REGION Network 2: +++ Werkingsmode Hand +++
   // Verwerking van de bedieningen van het aanraakscherm, en bepalen van de bedieningsmode Hand.
END_REGION

REGION Network 3: +++ Gewenste stand +++
   // Bepalen aan de hand van de actuele bediening of ontvangen sturing, wat de gewenste stand van de klep is.
END_REGION

REGION Network 4: +++ Klepsturing +++
   // Aansturen van de klep en terugmeldingsbewaking.
END_REGION

REGION Network 5: +++ Storingen +++
   // Verwerken van de storingsmeldingen.
END_REGION

REGION Network 6: Storing A001: Beveiliging aangesproken
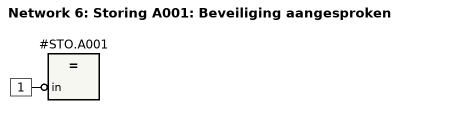
   #STO.A001 := NOT 1;
END_REGION

REGION Network 7 (SCL): EINDE
   // Variabelen van intern scada rakvlak naar outputs copieren
   #VAR_IF_KLG.STS_OPEN := #VAR.STS_OPEN;
   #VAR_IF_KLG.STS_TOE := #VAR.STS_TOE;
   #VAR_IF_KLG.STS_BEZ_OPEN := #VAR.STS_BEZ_OPEN;
   #VAR_IF_KLG.STS_BEZ_TOE := #VAR.STS_BEZ_TOE;
   #VAR_IF_KLG.BMO_HAND := #VAR.BMO_HAND;
   #VAR_IF_KLG.EXT_HW := #VAR.EXT_HW;
   #VAR_IF_KLG.STO := #STO;
END_REGION
END_FUNCTION_BLOCK

FUNCTION_BLOCK "TYPIC_C501_IF_KLH"   // FB63, FBD
TITLE = TYPIC_C501_IF_KLH: Handbediende klep
{ S7_Optimized_Access := 'TRUE' }
AUTHOR : OCOTECH
FAMILY : Typical
NAME : C501.704
// Logisch Object Besturing: C501.704
// 
// De interne functie handbediende klep verzorgt de bewaking van één van volgende componenten:
//  een handbediende klep
//  een leegzetvoorziening
//  een beo/ontluchtingsvoorziening
// stored: MemoryReserve 10, SetENOAutomatically false
   VAR_INPUT
      EXT_HW { ExternalAccessible := 'False'; ExternalVisible := 'False'; ExternalWritable := 'False'} : Bool;   // Sturings hardware (PLC) bewaking (1 = OK)
      IN_OPEN { ExternalAccessible := 'False'; ExternalVisible := 'False'; ExternalWritable := 'False'} : Bool;   // Handbediende klep is open
      IN_TOE { ExternalAccessible := 'False'; ExternalVisible := 'False'; ExternalWritable := 'False'} : Bool;   // Handbediende klep is toe
      CFG_OPEN { ExternalAccessible := 'False'; ExternalVisible := 'False'; ExternalWritable := 'False'} : Bool;   // Handbediende klep heeft een toestandsmelding Open
      CFG_TOE { ExternalAccessible := 'False'; ExternalVisible := 'False'; ExternalWritable := 'False'} : Bool;   // Handbediende klep heeft een toestandsmelding Toe
   END_VAR
   VAR_OUTPUT
      VAR_IF_KLH { ExternalAccessible := 'False'; ExternalVisible := 'False'; ExternalWritable := 'False'} : "C501_VAR_IF_KLH_TYPIC";   // Struct met alle variabelen naar bovenliggende functies
   END_VAR
   VAR
      STO { ExternalWritable := 'False'} : Struct   // Storingen
         A001 : Bool;   // Terugmeldingen Open en Dicht tegelijk
      END_STRUCT;
      VAR { ExternalWritable := 'False'} : Struct   // Variabelen
         STS_OPEN : Bool;   // Handbediende klep is open
         STS_TOE : Bool;   // Handbediende klep is toe
         EXT_HW { ExternalAccessible := 'False'; ExternalVisible := 'False'} : Bool;   // Sturings hardware (PLC) in storing
      END_STRUCT;
   END_VAR
BEGIN

REGION Network 1: START
END_REGION

REGION Network 2: +++ Status +++
   // De status van de handbediende klep (open / dicht) wordt doorgestuurd naar 3B.
END_REGION

REGION Network 3: +++ Storingen +++
   // Alle storingen worden doorgegeven aan 3B.
END_REGION

REGION Network 4: Storing A001: Terugmeldingen Open en Dicht tegelijk
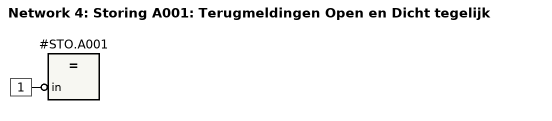
   #STO.A001 := NOT 1;
END_REGION

REGION Network 5 (SCL): EINDE
   // Variabelen van intern scada rakvlak naar outputs copieren
   #VAR_IF_KLH.STS_OPEN := #VAR.STS_OPEN;
   #VAR_IF_KLH.STS_TOE := #VAR.STS_TOE;
   #VAR_IF_KLH.EXT_HW := #VAR.EXT_HW;
   #VAR_IF_KLH.STO := #STO;
END_REGION
END_FUNCTION_BLOCK

FUNCTION_BLOCK "TYPIC_C501_IF_NME"   // FB62, FBD
TITLE = TYPIC_C501_IF_NME: Niveaumeting
{ S7_Optimized_Access := 'TRUE' }
AUTHOR : OCOTECH
FAMILY : Typical
NAME : C501.702
// Logisch Object Besturing: C501.702
// 
// De interne functie niveaumeting verzorgt de interne besturing en bewaking van een niveaumeting van de brandblusinstallatie.
// stored: MemoryReserve 10, SetENOAutomatically false
   VAR_INPUT
      EXT_HW { ExternalAccessible := 'False'; ExternalVisible := 'False'; ExternalWritable := 'False'} : Bool;   // Sturings hardware (PLC) bewaking (1 = OK)
      IN_MWA { ExternalAccessible := 'False'; ExternalVisible := 'False'; ExternalWritable := 'False'} : Word;   // Meetwaarde
      IN_HW { ExternalAccessible := 'False'; ExternalVisible := 'False'; ExternalWritable := 'False'} : Bool;   // Vlotter: 1 = Bovenwater / 0 = Onderwater
      IN_VHW { ExternalAccessible := 'False'; ExternalVisible := 'False'; ExternalWritable := 'False'} : Bool;   // Vlotter: 1 = Bovenwater / 0 = Onderwater
      IN_SD { ExternalAccessible := 'False'; ExternalVisible := 'False'; ExternalWritable := 'False'} : Bool;   // Vlotter: 1 = Bovenwater / 0 = Onderwater
      IN_SO { ExternalAccessible := 'False'; ExternalVisible := 'False'; ExternalWritable := 'False'} : Bool;   // Vlotter: 1 = Onderwater / 0 = Bovenwater
      IN_VRL { ExternalAccessible := 'False'; ExternalVisible := 'False'; ExternalWritable := 'False'} : Bool;   // Vlotter: 1 = Onderwater / 0 = Bovenwater
      IN_RL { ExternalAccessible := 'False'; ExternalVisible := 'False'; ExternalWritable := 'False'} : Bool;   // Vlotter: 1 = Onderwater / 0 = Bovenwater
      IN_AUT_C501 { ExternalAccessible := 'False'; ExternalVisible := 'False'; ExternalWritable := 'False'} : Bool;   // Beveiligingen: serie geschakelde terugmelding (1= OK)
      CFG_MAX { ExternalAccessible := 'False'; ExternalVisible := 'False'; ExternalWritable := 'False'} : Int;   // Waarde van input IN_MWA als maximum voor de scalering ter bepaling van NIV_MWA
      CFG_MIN { ExternalAccessible := 'False'; ExternalVisible := 'False'; ExternalWritable := 'False'} : Int;   // Waarde van input IN_MWA als minimum voor de scalering ter bepaling van NIV_MWA
      CFG_MAX_SWA { ExternalAccessible := 'False'; ExternalVisible := 'False'; ExternalWritable := 'False'} : Real;   // Waarde die toegekend wordt aan NIV_MWA als maximumwmaximumwaarde voor de meeteenheid
      CFG_MIN_SWA { ExternalAccessible := 'False'; ExternalVisible := 'False'; ExternalWritable := 'False'} : Real;   // Waarde die toegekend wordt aan NIV_MWA als minimumwmaximumwaarde voor de meeteenheid
   END_VAR
   VAR_OUTPUT
      VAR_IF_NME { ExternalAccessible := 'False'; ExternalVisible := 'False'; ExternalWritable := 'False'} : "C501_VAR_IF_NME_TYPIC";   // Struct met alle variabelen naar de basisfunctie
   END_VAR
   VAR
      STO { ExternalWritable := 'False'} : Struct   // Storingen
         A001 : Bool;   // Beveiliging aangesproken
         A002 : Bool;   // Draadbreuk analoge meting
         A003 : Bool;   // Meetbereik overschreden
         A004 : Bool;   // Status vlotters inconsistent
      END_STRUCT;
      VAR { ExternalWritable := 'False'} : Struct   // Variabelen
         MWA : Real;   // Meetwaarde
         HW : USInt;   // Hoogwater vlotter
         VHW : USInt;   // Voorwaarschuwing hoogwater
         SD : USInt;   // Suppletie dicht
         SO : USInt;   // Suppletie open
         VRL : USInt;   // Voorwaarschuwing reservoir leeg
         RL : USInt;   // Reservoir leeg
         EXT_HW { ExternalAccessible := 'False'; ExternalVisible := 'False'} : Bool;   // Sturings hardware (PLC) in storing
      END_STRUCT;
   END_VAR
BEGIN

REGION Network 1: START
END_REGION

REGION Network 2: +++ Bepalen status peilen (vlotters) +++
   // Aan de hand van de status van de vlotters (inputs) wordt het peil (onderwater/bovenwater) bepaalt.
END_REGION

REGION Network 3: +++ Meting +++
   // Verwerken van de analoge meting.
END_REGION

REGION Network 4: +++ Storingen +++
   // Verwerken van de storingsmeldingen.
END_REGION

REGION Network 5: Storing A001: Beveiliging aangesproken
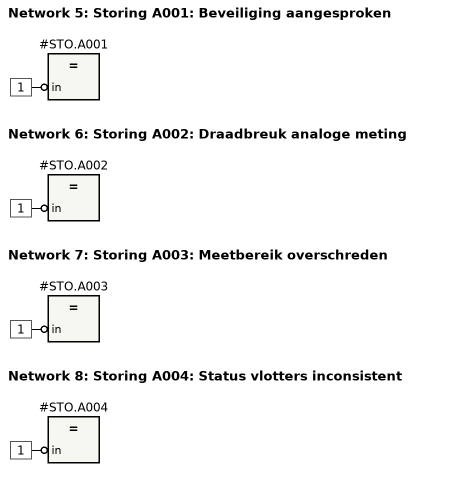
   #STO.A001 := NOT 1;
END_REGION

REGION Network 6: Storing A002: Draadbreuk analoge meting
   #STO.A002 := NOT 1;
END_REGION

REGION Network 7: Storing A003: Meetbereik overschreden
   #STO.A003 := NOT 1;
END_REGION

REGION Network 8: Storing A004: Status vlotters inconsistent
   #STO.A004 := NOT 1;
END_REGION

REGION Network 9 (SCL): EINDE
   // Variabelen van intern scada rakvlak naar outputs copieren
   #VAR_IF_NME.MWA := #VAR.MWA;
   #VAR_IF_NME.HW := #VAR.HW;
   #VAR_IF_NME.VHW := #VAR.VHW;
   #VAR_IF_NME.SD := #VAR.SD;
   #VAR_IF_NME.SO := #VAR.SO;
   #VAR_IF_NME.VRL := #VAR.VRL;
   #VAR_IF_NME.RL := #VAR.RL;
   #VAR_IF_NME.EXT_HW := #VAR.EXT_HW;
   #VAR_IF_NME.STO := #STO;
END_REGION
END_FUNCTION_BLOCK

FUNCTION_BLOCK "TYPIC_C501_IF_SME"   // FB61, FBD
TITLE = TYPIC_C501_IF_SME: Debietmeting
{ S7_Optimized_Access := 'TRUE' }
AUTHOR : OCOTECH
FAMILY : Typical
NAME : C501.711
// Logisch Object Besturing: C501.711
// 
// De interne functie debietmeting verzorgt de interne besturing en bewaking van een debietmeting.
// stored: MemoryReserve 10, SetENOAutomatically false
   VAR_INPUT
      EXT_HW { ExternalAccessible := 'False'; ExternalVisible := 'False'; ExternalWritable := 'False'} : Bool;   // Sturings hardware (PLC) bewaking (1 = OK)
      IN_MWA { ExternalAccessible := 'False'; ExternalVisible := 'False'; ExternalWritable := 'False'} : Word;   // Meetwaarde
      IN_STO { ExternalAccessible := 'False'; ExternalVisible := 'False'; ExternalWritable := 'False'} : Bool;   // Storing (1= OK)
      IN_AUT_C501 { ExternalAccessible := 'False'; ExternalVisible := 'False'; ExternalWritable := 'False'} : Bool;   // Beveiligingen: serie geschakelde terugmelding (1= OK)
      CFG_MAX_SWA { ExternalAccessible := 'False'; ExternalVisible := 'False'; ExternalWritable := 'False'} : Real;   // Maximale waarde debietmeting
   END_VAR
   VAR_OUTPUT
      VAR_IF_SME { ExternalAccessible := 'False'; ExternalVisible := 'False'; ExternalWritable := 'False'} : "C501_VAR_IF_SME_TYPIC";   // Struct met alle variabelen naar bovenliggende functies
   END_VAR
   VAR
      STO { ExternalWritable := 'False'} : Struct   // Storingen
         A001 : Bool;   // Beveiliging aangesproken
         A002 : Bool;   // Draadbreuk analoge meting
         A003 : Bool;   // Meetbereik overschreden
         A004 : Bool;   // Debietmeter geeft storing
      END_STRUCT;
      VAR { ExternalWritable := 'False'} : Struct   // Variabelen
         MWA : Real;   // Meetwaarde
         EXT_HW { ExternalAccessible := 'False'; ExternalVisible := 'False'} : Bool;   // Sturings hardware (PLC) in storing
      END_STRUCT;
   END_VAR
BEGIN

REGION Network 1: START
END_REGION

REGION Network 2: +++ Verwerking analoge meting +++
   // Verwerking analoge meting naar een meetwaarde in m3/u en detectie storingen van de meting.
END_REGION

REGION Network 3: +++ Storingen +++
   // Storingen van de analoge meting.
END_REGION

REGION Network 4: Storing A001: Beveiliging aangesproken
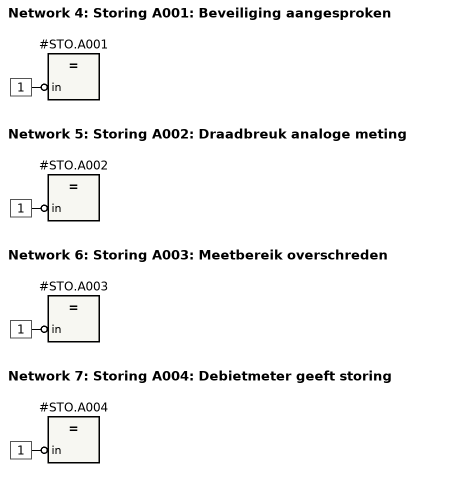
   #STO.A001 := NOT 1;
END_REGION

REGION Network 5: Storing A002: Draadbreuk analoge meting
   #STO.A002 := NOT 1;
END_REGION

REGION Network 6: Storing A003: Meetbereik overschreden
   #STO.A003 := NOT 1;
END_REGION

REGION Network 7: Storing A004: Debietmeter geeft storing
   #STO.A004 := NOT 1;
END_REGION

REGION Network 8 (SCL): EINDE
   // Variabelen van intern scada rakvlak naar outputs copieren
   #VAR_IF_SME.MWA := #VAR.MWA;
   #VAR_IF_SME.EXT_HW := #VAR.EXT_HW;
   #VAR_IF_SME.STO := #STO;
END_REGION
END_FUNCTION_BLOCK

FUNCTION_BLOCK "TYPIC_C501_IF_TME"   // FB60, FBD
TITLE = TYPIC_C501_IF_TME: Temperatuurmeting
{ S7_Optimized_Access := 'TRUE' }
AUTHOR : OCOTECH
FAMILY : Typical
NAME : C501.712
// Logisch Object Besturing: C501.712
// 
// De interne functie temperatuurmeting verzorgt de interne besturing en bewaking van een temperatuurmeting.
// stored: MemoryReserve 10, SetENOAutomatically false
   VAR_INPUT
      EXT_HW { ExternalAccessible := 'False'; ExternalVisible := 'False'; ExternalWritable := 'False'} : Bool;   // Sturings hardware (PLC) bewaking (1 = OK)
      IN_MWA { ExternalAccessible := 'False'; ExternalVisible := 'False'; ExternalWritable := 'False'} : Word;   // Meetwaarde
      IN_AUT_C501 { ExternalAccessible := 'False'; ExternalVisible := 'False'; ExternalWritable := 'False'} : Bool;   // Beveiligingen: serie geschakelde terugmelding (1= OK)
      CFG_MAX_SWA { ExternalAccessible := 'False'; ExternalVisible := 'False'; ExternalWritable := 'False'} : Real;   // Maximale waarde temperatuurmeting
      CFG_MIN_SWA { ExternalAccessible := 'False'; ExternalVisible := 'False'; ExternalWritable := 'False'} : Real;   // Minimale waarde temperatuurmeting
   END_VAR
   VAR_OUTPUT
      VAR_IF_TME { ExternalAccessible := 'False'; ExternalVisible := 'False'; ExternalWritable := 'False'} : "C501_VAR_IF_TME_TYPIC";   // Struct met alle variabelen naar bovenliggende functies
   END_VAR
   VAR
      STO { ExternalWritable := 'False'} : Struct   // Storingen
         A001 : Bool;   // Beveiliging aangesproken
         A002 : Bool;   // Draadbreuk analoge meting
         A003 : Bool;   // Meetbereik overschreden
         A004 : Bool;   // Temperatuurmeter geeft storing
      END_STRUCT;
      VAR { ExternalWritable := 'False'} : Struct   // Variabelen
         MWA : Real;   // Meetwaarde
         EXT_HW { ExternalAccessible := 'False'; ExternalVisible := 'False'} : Bool;   // Sturings hardware (PLC) in storing
      END_STRUCT;
   END_VAR
BEGIN

REGION Network 1: START
END_REGION

REGION Network 2: +++ Verwerking analoge meting +++
   // Verwerking analoge meting naar een meetwaarde in m3/u en detectie storingen van de meting.
END_REGION

REGION Network 3: +++ Storingen +++
   // Storingen van de analoge meting.
END_REGION

REGION Network 4: Storing A001: Beveiliging aangesproken
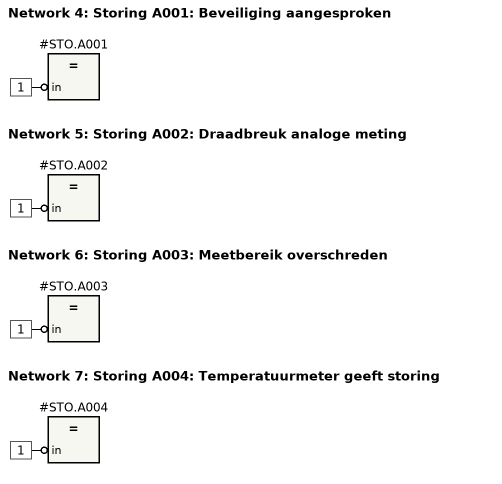
   #STO.A001 := NOT 1;
END_REGION

REGION Network 5: Storing A002: Draadbreuk analoge meting
   #STO.A002 := NOT 1;
END_REGION

REGION Network 6: Storing A003: Meetbereik overschreden
   #STO.A003 := NOT 1;
END_REGION

REGION Network 7: Storing A004: Temperatuurmeter geeft storing
   #STO.A004 := NOT 1;
END_REGION

REGION Network 8 (SCL): EINDE
   // Variabelen van intern scada rakvlak naar outputs copieren
   #VAR_IF_TME.MWA := #VAR.MWA;
   #VAR_IF_TME.EXT_HW := #VAR.EXT_HW;
   #VAR_IF_TME.STO := #STO;
END_REGION
END_FUNCTION_BLOCK

FUNCTION_BLOCK "TYPIC_C501_IF_TRA"   // FB59, FBD
TITLE = TYPIC_C501_IF_TRA: Tracing
{ S7_Optimized_Access := 'TRUE' }
AUTHOR : OCOTECH
FAMILY : Typical
NAME : C501.705
// Logisch Object Besturing: C501.705
// stored: MemoryReserve 10, SetENOAutomatically false
   VAR_INPUT
      EXT_HW { ExternalAccessible := 'False'; ExternalVisible := 'False'; ExternalWritable := 'False'} : Bool;   // Sturings hardware (PLC) bewaking (1 = OK)
      IN_STO { ExternalAccessible := 'False'; ExternalVisible := 'False'; ExternalWritable := 'False'} : Bool;   // Storing Tracing (1 = OK)
   END_VAR
   VAR_OUTPUT
      VAR_IF_TRA { ExternalAccessible := 'False'; ExternalVisible := 'False'; ExternalWritable := 'False'} : "C501_VAR_IF_TRA_TYPIC";   // Struct met alle variabelen naar bovenliggende functies
   END_VAR
   VAR
      STO { ExternalWritable := 'False'} : Struct   // Storingen
         A001 : Bool;   // Storing vorstbeveiliging
      END_STRUCT;
      VAR { ExternalWritable := 'False'} : Struct   // Variabelen
         EXT_HW { ExternalAccessible := 'False'; ExternalVisible := 'False'} : Bool;   // Sturings hardware (PLC) in storing
      END_STRUCT;
   END_VAR
BEGIN

REGION Network 1: START
END_REGION

REGION Network 2: +++ Storingen +++
   // Verwerken van de storingsmeldingen (inputs).
END_REGION

REGION Network 3: Storing A001: Storing vorstbeveiliging
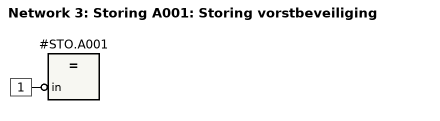
   #STO.A001 := NOT 1;
END_REGION

REGION Network 4 (SCL): EINDE
   // Variabelen van intern scada rakvlak naar outputs copieren
   #VAR_IF_TRA.EXT_HW := #VAR.EXT_HW;
   #VAR_IF_TRA.STO := #STO;
END_REGION
END_FUNCTION_BLOCK

FUNCTION_BLOCK "TYPIC_C501_SF_DME"   // FB55, FBD
TITLE = TYPIC_C501_SF_DME: Drukmeting
{ S7_Optimized_Access := 'TRUE' }
AUTHOR : OCOTECH
FAMILY : Typical
NAME : C501.813
// Logisch Object Besturing: C501.813
// 
// Het doel van deze subfunctie is om de algemene sturing en bediening vanuit 3B te voorzien van een drukmeting behorende tot de brandblusinstallatie.
// stored: MemoryReserve 10, SetENOAutomatically false
   VAR_INPUT
      CFG_SIG_HH { ExternalAccessible := 'False'; ExternalVisible := 'False'; ExternalWritable := 'False'} : Real;   // Schakeldrempel signalering te hoog
      CFG_SIG_H { ExternalAccessible := 'False'; ExternalVisible := 'False'; ExternalWritable := 'False'} : Real;   // Schakeldrempel signalering voorwaarschuwing hoog
      CFG_HYS_H { ExternalAccessible := 'False'; ExternalVisible := 'False'; ExternalWritable := 'False'} : Real;   // Hysteresis op signalering te hoog en voorwaarschuwing hoog
      CFG_ITYD_H { ExternalAccessible := 'False'; ExternalVisible := 'False'; ExternalWritable := 'False'} : Real;   // Tijdsvertraging signalering te hoog
      CFG_SIG_L { ExternalAccessible := 'False'; ExternalVisible := 'False'; ExternalWritable := 'False'} : Real;   // Schakeldrempel signalering te laag
      CFG_HYS_L { ExternalAccessible := 'False'; ExternalVisible := 'False'; ExternalWritable := 'False'} : Real;   // Hysteresis op signalering te laag
      CFG_ITYD_L { ExternalAccessible := 'False'; ExternalVisible := 'False'; ExternalWritable := 'False'} : Time;   // Tijdsvertraging signalering te laag
   END_VAR
   VAR_OUTPUT
      VAR_DME { ExternalAccessible := 'False'; ExternalVisible := 'False'; ExternalWritable := 'False'} : "C501_VAR_DME_TYPIC";   // Struct met alle variabelen van de drukmeting
   END_VAR
   VAR_IN_OUT
      STU_DME : "C501_STU_DME_TYPIC";   // Struct met alle sturingen vanuit de bovenliggende functie
      VAR_IF_DME : "C501_VAR_IF_DME_TYPIC";   // Struct met alle variabelen vanuit de interne sturing
   END_VAR
   VAR
      BED : Struct   // Bedieningen
         OBS : Struct   // Activeer of deactiveer de detectie van de stand van de deur van de hydrantkast
            X : "UDT_BED_ALG";
            KNOP { S7_SetPoint := 'True'} : Array[0..1] of "UDT_BED_KNOP";
         END_STRUCT;
      END_STRUCT;
      BED_OBS { ExternalWritable := 'False'} : "TYPIC_HF_BED_ALG_KNOP";   // Activeer of deactiveer de detectie van de stand van de deur van de hydrantkast
      SIG { ExternalWritable := 'False'} : Struct   // Signaleringen
         AA01 : Bool;   // Drukmeting niet observeerbaar
         AA02 : Bool;   // Storing algemeen
         AA03 : Bool;   // Druk te laag
         AA04 : Bool;   // Voorwaarschuwing druk hoog
         AA05 : Bool;   // Druk te hoog
         A001 : Bool;   // Beveiliging aangesproken
         A002 : Bool;   // Draadbreuk analoge meting
         A003 : Bool;   // Meetbereik overschreden
      END_STRUCT;
      VAR { ExternalWritable := 'False'} : Struct   // Variabelen
         RNO : USInt;   // Reden niet observeerbaar
         AUT : USInt;   // Beveiliging aangesproken
         MWA : USInt;   // Meetwaarde
         OBS { ExternalAccessible := 'False'; ExternalVisible := 'False'} : USInt;   // Observeerbaarheid
      END_STRUCT;
      HF_BST_OBS { ExternalAccessible := 'False'; ExternalVisible := 'False'; ExternalWritable := 'False'} : "TYPIC_HF_BST_OBS";   // Hulp functie besturing
   END_VAR
   // // BED.OBS.KNOP[0] : InDienst
   // // BED.OBS.KNOP[1] : UitDienst
BEGIN

REGION Network 1: START
END_REGION

REGION Network 2: +++ Bedieningen +++
   // Vrijgave en verwerking van de bedieningen (centrale en lokale bediening). De bedienwaardes worden daarna in de verdere deelfunctionaliteiten gebruikt.
END_REGION

REGION Network 3: Knoppen BED_OBS(Activeer of deactiveer de detectie van de stand van de deur van de hydrantkast)
   // Waardes en vrijge van de knoppen BED_OBS
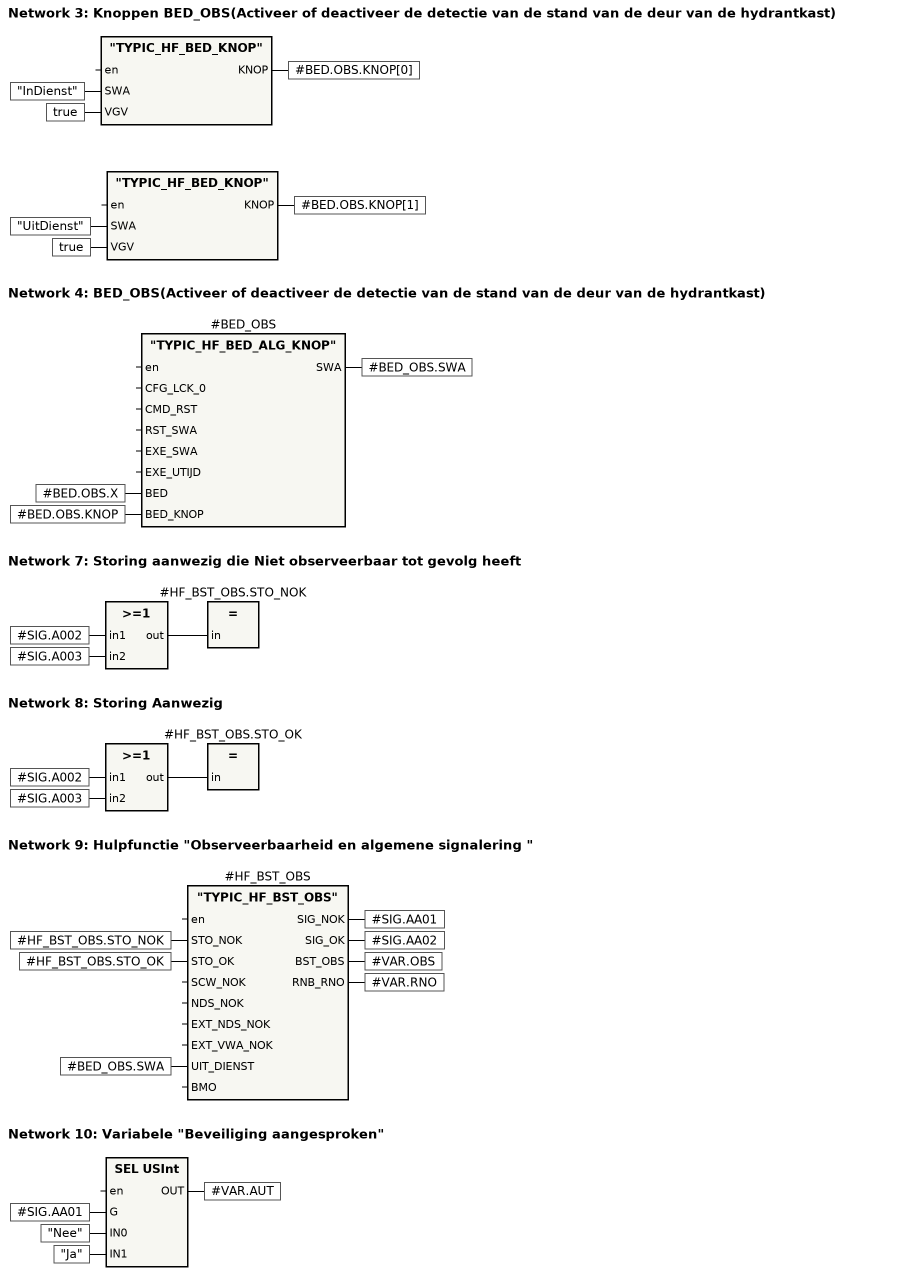
   "TYPIC_HF_BED_KNOP"(SWA := "InDienst", VGV := true, KNOP => #BED.OBS.KNOP[0]);
   "TYPIC_HF_BED_KNOP"(SWA := "UitDienst", VGV := true, KNOP => #BED.OBS.KNOP[1]);
END_REGION

REGION Network 4: BED_OBS(Activeer of deactiveer de detectie van de stand van de deur van de hydrantkast)
   // Verwerking BED_OBS
   #BED_OBS(BED := #BED.OBS.X, BED_KNOP := #BED.OBS.KNOP, SWA => #BED_OBS.SWA);   // "TYPIC_HF_BED_ALG_KNOP"
END_REGION

REGION Network 5: +++ Verwerking meetwaarde en statussen +++
   // De meetwaarde en de status wordt ontvangen vanuit de interne sturing van de drukmeting.
END_REGION

REGION Network 6: +++ Signaleringen en observeerbaarheid +++
   // Aanmaken signaleringen, bepalen observeerbaarheid (observeerbaar / niet observeerbaar) en bepalen reden niet observeerbaar.
END_REGION

REGION Network 7: Storing aanwezig die Niet observeerbaar tot gevolg heeft
   // OR-verknoping van alle storingen om input STO_BST_NOK van de hulpfunctie "Observeerbaarheid en algemene signlaring"
   #HF_BST_OBS.STO_NOK := #SIG.A002 OR #SIG.A003;
END_REGION

REGION Network 8: Storing Aanwezig
   // OR-verknoping van alle storingen om input STO_BST_OK van de hulpfunctie "Observeerbaarheid en algemene signlaring"
   #HF_BST_OBS.STO_OK := #SIG.A002 OR #SIG.A003;
END_REGION

REGION Network 9: Hulpfunctie "Observeerbaarheid en algemene signalering "
   // Bepalen variabele "Observeerbaarheid" en "reden niet Observeerbaarheid", Signaleringen "Observeerbaarheid" en "algmene storing".
   #HF_BST_OBS(STO_NOK := #HF_BST_OBS.STO_NOK,   // "TYPIC_HF_BST_OBS"
               STO_OK := #HF_BST_OBS.STO_OK,
               UIT_DIENST := #BED_OBS.SWA,
               SIG_NOK => #SIG.AA01,
               SIG_OK => #SIG.AA02,
               BST_OBS => #VAR.OBS,
               RNB_RNO => #VAR.RNO);
END_REGION

REGION Network 10: Variabele "Beveiliging aangesproken"
   // De variabele VAR_AUT geef aan of er een beveilliging aangesproken is. Deze variabele laat toe dat de verkeersoperator op SCADA kan zien of er een beveilliging aangesproken is voor deze component.
   #VAR.AUT := SEL(G := #SIG.AA01, IN0 := "Nee", IN1 := "Ja");
END_REGION

REGION Network 11 (SCL): EINDE
   // Variabelen van intern scada rakvlak naar outputs copieren
   #VAR_DME.MWA := #VAR.MWA;
   #VAR_DME.OBS := #VAR.OBS;
END_REGION
END_FUNCTION_BLOCK

FUNCTION_BLOCK "TYPIC_C501_SF_TME"   // FB46, FBD
TITLE = TYPIC_C501_SF_TME: Temperatuurmeting
{ S7_Optimized_Access := 'TRUE' }
AUTHOR : OCOTECH
FAMILY : Typical
NAME : C501.815
// Logisch Object Besturing: C501.815
// 
// Het doel van deze subfunctie is om de algemene sturing en bediening vanuit 3B te voorzien van een temperatuurmeting behorende tot de brandblusinstallatie.
// stored: MemoryReserve 10, SetENOAutomatically false
   VAR_INPUT
      CFG_SIG_L { ExternalAccessible := 'False'; ExternalVisible := 'False'; ExternalWritable := 'False'} : Real;   // Schakeldrempel signalering te laag
      CFG_HYS_L { ExternalAccessible := 'False'; ExternalVisible := 'False'; ExternalWritable := 'False'} : Real;   // Hysteresis op signalering te laag
      CFG_ITYD_L { ExternalAccessible := 'False'; ExternalVisible := 'False'; ExternalWritable := 'False'} : Time;   // Tijdsvertraging signalering te laag
   END_VAR
   VAR_OUTPUT
      VAR_TME { ExternalAccessible := 'False'; ExternalVisible := 'False'; ExternalWritable := 'False'} : "C501_VAR_TME_TYPIC";   // Struct met alle variabelen van de temperatuurmeting
   END_VAR
   VAR_IN_OUT
      STU_TME : "C501_STU_TME_TYPIC";   // Struct met alle sturingen vanuit de bovenliggende functie
      VAR_IF_TME : "C501_VAR_IF_TME_TYPIC";   // Struct met alle variabelen vanuit de interne sturing
   END_VAR
   VAR
      BED : Struct   // Bedieningen
         OBS : Struct   // Activeer of deactiveer de detectie van de stand van de deur van de hydrantkast
            X : "UDT_BED_ALG";
            KNOP { S7_SetPoint := 'True'} : Array[0..1] of "UDT_BED_KNOP";
         END_STRUCT;
      END_STRUCT;
      BED_OBS { ExternalWritable := 'False'} : "TYPIC_HF_BED_ALG_KNOP";   // Activeer of deactiveer de detectie van de stand van de deur van de hydrantkast
      SIG { ExternalWritable := 'False'} : Struct   // Signaleringen
         AA01 : Bool;   // Temperatuurmeting niet observeerbaar
         AA02 : Bool;   // Storing algemeen
         AA03 : Bool;   // Temperatuur te laag
         A001 : Bool;   // Beveiliging aangesproken
         A002 : Bool;   // Draadbreuk analoge meting
         A003 : Bool;   // Meetbereik overschreden
      END_STRUCT;
      VAR { ExternalWritable := 'False'} : Struct   // Variabelen
         RNO : USInt;   // Reden niet observeerbaar
         AUT : USInt;   // Beveiliging aangesproken
         MWA : USInt;   // Meetwaarde
         OBS { ExternalAccessible := 'False'; ExternalVisible := 'False'} : USInt;   // Observeerbaarheid
      END_STRUCT;
      HF_BST_OBS { ExternalAccessible := 'False'; ExternalVisible := 'False'; ExternalWritable := 'False'} : "TYPIC_HF_BST_OBS";   // Hulp functie besturing
   END_VAR
   // // BED.OBS.KNOP[0] : InDienst
   // // BED.OBS.KNOP[1] : UitDienst
BEGIN

REGION Network 1: START
END_REGION

REGION Network 2: +++ Bedieningen +++
   // Vrijgave en verwerking van de bedieningen (centrale en lokale bediening). De bedienwaardes worden daarna in de verdere deelfunctionaliteiten gebruikt.
END_REGION

REGION Network 3: Knoppen BED_OBS(Activeer of deactiveer de detectie van de stand van de deur van de hydrantkast)
   // Waardes en vrijge van de knoppen BED_OBS
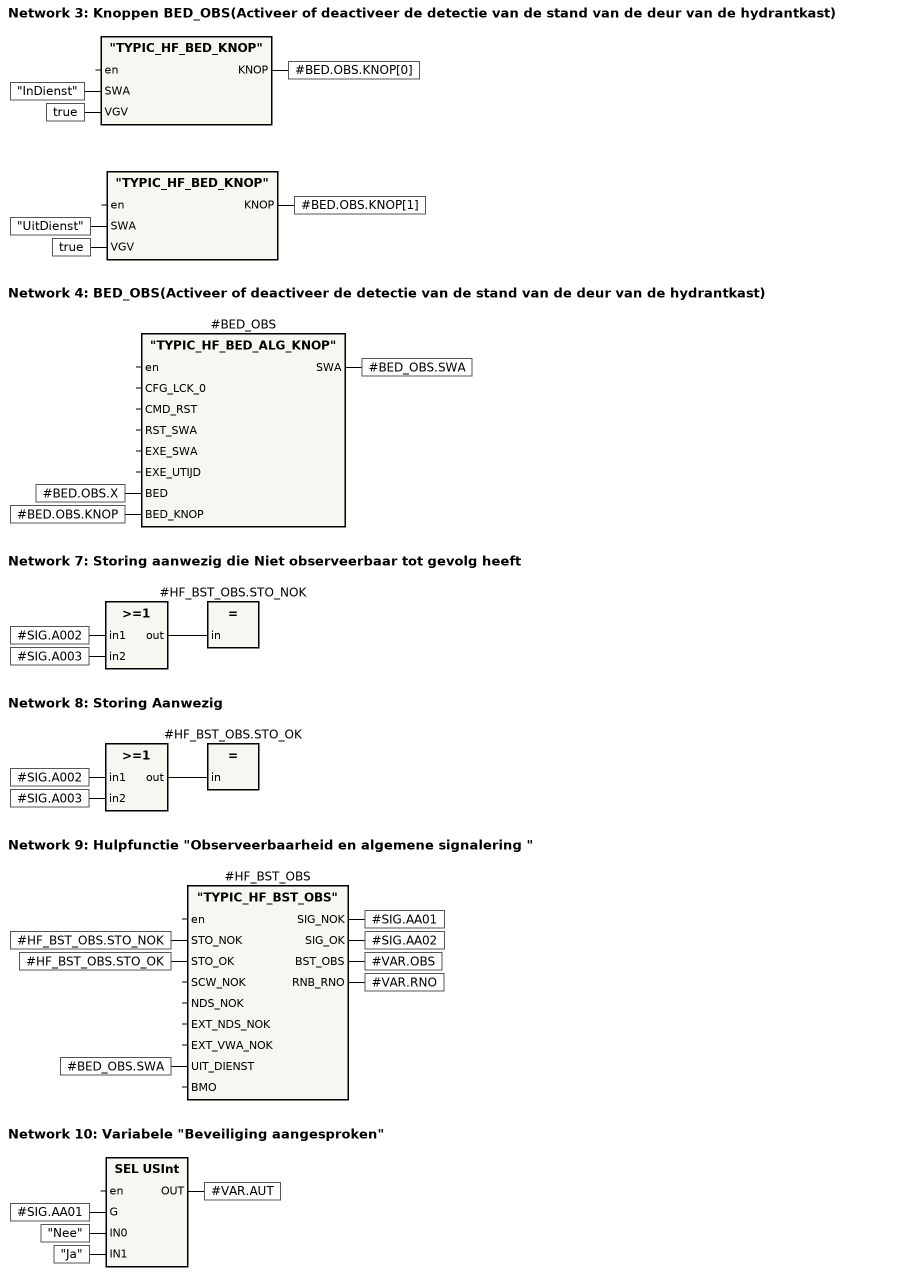
   "TYPIC_HF_BED_KNOP"(SWA := "InDienst", VGV := true, KNOP => #BED.OBS.KNOP[0]);
   "TYPIC_HF_BED_KNOP"(SWA := "UitDienst", VGV := true, KNOP => #BED.OBS.KNOP[1]);
END_REGION

REGION Network 4: BED_OBS(Activeer of deactiveer de detectie van de stand van de deur van de hydrantkast)
   // Verwerking BED_OBS
   #BED_OBS(BED := #BED.OBS.X, BED_KNOP := #BED.OBS.KNOP, SWA => #BED_OBS.SWA);   // "TYPIC_HF_BED_ALG_KNOP"
END_REGION

REGION Network 5: +++ Verwerking meetwaarde en statussen +++
   // De meetwaarde en de status wordt ontvangen vanuit de interne sturing van de temperatuurmeting.
END_REGION

REGION Network 6: +++ Signaleringen en observeerbaarheid +++
   // Aanmaken signaleringen, bepalen observeerbaarheid (observeerbaar / niet observeerbaar) en bepalen reden niet observeerbaar.
END_REGION

REGION Network 7: Storing aanwezig die Niet observeerbaar tot gevolg heeft
   // OR-verknoping van alle storingen om input STO_BST_NOK van de hulpfunctie "Observeerbaarheid en algemene signlaring"
   #HF_BST_OBS.STO_NOK := #SIG.A002 OR #SIG.A003;
END_REGION

REGION Network 8: Storing Aanwezig
   // OR-verknoping van alle storingen om input STO_BST_OK van de hulpfunctie "Observeerbaarheid en algemene signlaring"
   #HF_BST_OBS.STO_OK := #SIG.A002 OR #SIG.A003;
END_REGION

REGION Network 9: Hulpfunctie "Observeerbaarheid en algemene signalering "
   // Bepalen variabele "Observeerbaarheid" en "reden niet Observeerbaarheid", Signaleringen "Observeerbaarheid" en "algmene storing".
   #HF_BST_OBS(STO_NOK := #HF_BST_OBS.STO_NOK,   // "TYPIC_HF_BST_OBS"
               STO_OK := #HF_BST_OBS.STO_OK,
               UIT_DIENST := #BED_OBS.SWA,
               SIG_NOK => #SIG.AA01,
               SIG_OK => #SIG.AA02,
               BST_OBS => #VAR.OBS,
               RNB_RNO => #VAR.RNO);
END_REGION

REGION Network 10: Variabele "Beveiliging aangesproken"
   // De variabele VAR_AUT geef aan of er een beveilliging aangesproken is. Deze variabele laat toe dat de verkeersoperator op SCADA kan zien of er een beveilliging aangesproken is voor deze component.
   #VAR.AUT := SEL(G := #SIG.AA01, IN0 := "Nee", IN1 := "Ja");
END_REGION

REGION Network 11 (SCL): EINDE
   // Variabelen van intern scada rakvlak naar outputs copieren
   #VAR_TME.MWA := #VAR.MWA;
   #VAR_TME.OBS := #VAR.OBS;
END_REGION
END_FUNCTION_BLOCK

FUNCTION_BLOCK "TYPIC_C904_BF_SPI"   // FB44, FBD
TITLE = TYPIC_C904_BF_SPI: Schoonvloeistofpompinstallatie
{ S7_Optimized_Access := 'TRUE' }
AUTHOR : OCOTECH
FAMILY : Typical
NAME : C904.801
// Logisch Object Besturing: C904.801
// 
// 								Het doel van de BF SPI (schoonvloeistofpompinstallatie) is om de
// 								algemene sturing te voorzien van de schoonvloeistofpompinstallatie.
// 								De algemene sturing omvat het weergeven van de algemene toestand en
// 								het aano en afschakelen van pompen in functie van het vloeistofpeil
// 								en het actieve regime.
// stored: MemoryReserve 10, SetENOAutomatically false
   VAR_INPUT
      CFG_TST_UTYD { ExternalAccessible := 'False'; ExternalVisible := 'False'; ExternalWritable := 'False'} : Time;   // Time-out standverandering pompinstallatie (transitiestatus onbereikt)
      CFG_TST_OK_TYD { ExternalAccessible := 'False'; ExternalVisible := 'False'; ExternalWritable := 'False'} : Time;   // Stabilisatietijd voor de toestand OK (bereikt)
      CFG_NIV_H { ExternalAccessible := 'False'; ExternalVisible := 'False'; ExternalWritable := 'False'} : Real;   // Grenswaarde voor dreigende overloop (minder dan 30m3 bergruimte)
      CFG_NIV_HH { ExternalAccessible := 'False'; ExternalVisible := 'False'; ExternalWritable := 'False'} : Real;   // Grenswaarde voor overloop
      CFG_NIV_ITYD { ExternalAccessible := 'False'; ExternalVisible := 'False'; ExternalWritable := 'False'} : Time;   // Inschakelvertraging storingen grenswaarde
      CFG_NIV_HYS { ExternalAccessible := 'False'; ExternalVisible := 'False'; ExternalWritable := 'False'} : Real;   // Hysteresis storingen grenswaarde
      CFG_DEB_H { ExternalAccessible := 'False'; ExternalVisible := 'False'; ExternalWritable := 'False'} : Real;   // Grenswaarde minimaal debiet bij 1 aangeschakelde pomp
      CFG_DEB_HH { ExternalAccessible := 'False'; ExternalVisible := 'False'; ExternalWritable := 'False'} : Real;   // Grenswaarde minimaal debiet bij meerdere aangeschakelde pompen
      CFG_ITYD_DEB { ExternalAccessible := 'False'; ExternalVisible := 'False'; ExternalWritable := 'False'} : Time;   // Tijdsvertraging voor alarm afvoer verstopt (pomp aangeschakeld en minimaal debiet niet bereikt)
      STU_CMD_AUT { ExternalAccessible := 'False'; ExternalVisible := 'False'; ExternalWritable := 'False'} : USInt;   // Groepscommando: schakel in automatisch
      STU_CMD_WRE { ExternalAccessible := 'False'; ExternalVisible := 'False'; ExternalWritable := 'False'} : USInt;   // Sturing regime
      STU_ALG_LCK_SIG { ExternalAccessible := 'False'; ExternalVisible := 'False'; ExternalWritable := 'False'} : USInt;   // Onderdruk alarmen
   END_VAR
   VAR_OUTPUT
      VAR_PWR { ExternalAccessible := 'False'; ExternalVisible := 'False'; ExternalWritable := 'False'} : Real;   // Som actuele vermogens van alle pompen
      STU_PMP1 { ExternalAccessible := 'False'; ExternalVisible := 'False'; ExternalWritable := 'False'} : USInt;   // Sturing pomp
      STU_PMP2 { ExternalAccessible := 'False'; ExternalVisible := 'False'; ExternalWritable := 'False'} : USInt;   // Sturing pomp
      STU_PMP3 { ExternalAccessible := 'False'; ExternalVisible := 'False'; ExternalWritable := 'False'} : USInt;   // Sturing pomp
      STU_IF_SPI { ExternalAccessible := 'False'; ExternalVisible := 'False'; ExternalWritable := 'False'} : USInt;   // Gewenst regime (naar interne sturing)
   END_VAR
   VAR_IN_OUT
      VAR_IF_SPI : "C904_VAR_IF_SPI_TYPIC";   // Struct met variabelen ontvangen van de interne sturing van de pompinstallatie
      VAR_PMP : Array[*] of "C904_VAR_PMP_TYPIC";   // Array met alle pompen, met alle variabelen van de pomp
      VAR_NIV : "C904_VAR_NIV_TYPIC";   // Struct met alle variabelen ontvangen van de subfunctie niveaumeting
      VAR_DEB : "C904_VAR_DEB_TYPIC";   // Struct met alle variabelen ontvangen van de subfunctie debietmeting
   END_VAR
   VAR
      BED : Struct   // Bedieningen
         ALG : Struct   // Gewenste stand
            X : "UDT_BED_ALG";
            KNOP { S7_SetPoint := 'True'} : Array[0..3] of "UDT_BED_KNOP";
         END_STRUCT;
      END_STRUCT;
      BED_ALG { ExternalWritable := 'False'} : "TYPIC_HF_BED_ALG_KNOP";   // Gewenste stand
      SIG { ExternalWritable := 'False'} : Struct   // Signaleringen
         AA01 : Bool;   // Gewenste stand niet bereikt (transitiestatus = niet bereikt)
         AA02 : Bool;   // Schoonvloeistofpompinstallatie dreigt over te lopen
         AA03 : Bool;   // Overschrijding capaciteit schoonvloeistofpompinstallatie (overloop)
         AA04 : Bool;   // Afvoer verstopt en dreiging overloop van de schoonvloeistofpompinstallatie
         AA05 : Bool;   // Afvoer verstopt
         AB01 : Bool;   // Schoonvloeistofpompinstallatie niet beschikbaar
         AB02 : Bool;   // Schoonvloeistofpompinstallatie beperkt beschikbaar
         A001 : Bool;   // Beveiliging aangesproken
         A002 : Bool;   // Beveiliging No-Break aangesproken
         A003 : Bool;   // Overspanningsbeveiliging aangesproken
         A004 : Bool;   // Schuif ALSB uitgeschakeld
         A005 : Bool;   // Schuif ALSB in test
         A006 : Bool;   // Schuif ALSB uitgereden
         A007 : Bool;   // Nisdeur niet gesloten
         A008 : Bool;   // Storing tracing
      END_STRUCT;
      VAR { ExternalWritable := 'False'} : Struct   // Variabelen
         BSC : USInt;   // Geeft de beschikbaarheid aan van het deelsysteem
         TST_BWA : USInt;   // De status van de transitie van het deelsysteem
         BMO : USInt;   // Bedieningsmode
         WRE_BWA : USInt;   // Actueel regime
         CAPA : USInt;   // Beschikbare pompcapaciteit
         STS_TRA : USInt;   // Status van de tracing
         STS_NIV : USInt;   // Vloeistofniveau bepaald door de stand van de vlotters
         WRE_SWA { ExternalAccessible := 'False'; ExternalVisible := 'False'} : USInt;   // Gewenst regime
         REQ_AAN { ExternalAccessible := 'False'; ExternalVisible := 'False'} : USInt;   // Gewenst aantal aangeschakelde pompen
         CAPA_OK { ExternalAccessible := 'False'; ExternalVisible := 'False'} : USInt;   // Aantal beschikbare pompen
         STS_AAN { ExternalAccessible := 'False'; ExternalVisible := 'False'} : USInt;   // Actueel aantal aangeschakelde pompen
      END_STRUCT;
      HF_TST { ExternalAccessible := 'False'; ExternalVisible := 'False'; ExternalWritable := 'False'} : "TYPIC_HF_TST";   // Hulpfunctie transitiestatus
   END_VAR
   // // BED.ALG.KNOP[0] : Auto
   // // BED.ALG.KNOP[1] : Leeghouden
   // // BED.ALG.KNOP[2] : Bergen
   // // BED.ALG.KNOP[3] : Uit
BEGIN

REGION Network 1: START
END_REGION

REGION Network 2: +++ Bedieningen +++
   // Vrijgave en verwerking van de bedieningen (centrale en
   // 										lokale bediening). De bedienwaardes worden daarna in de
   // 										verdere deelfunctionaliteiten gebruikt.
END_REGION

REGION Network 3: Knoppen BED_ALG(Gewenste stand)
   // Waardes en vrijge van de knoppen BED_ALG
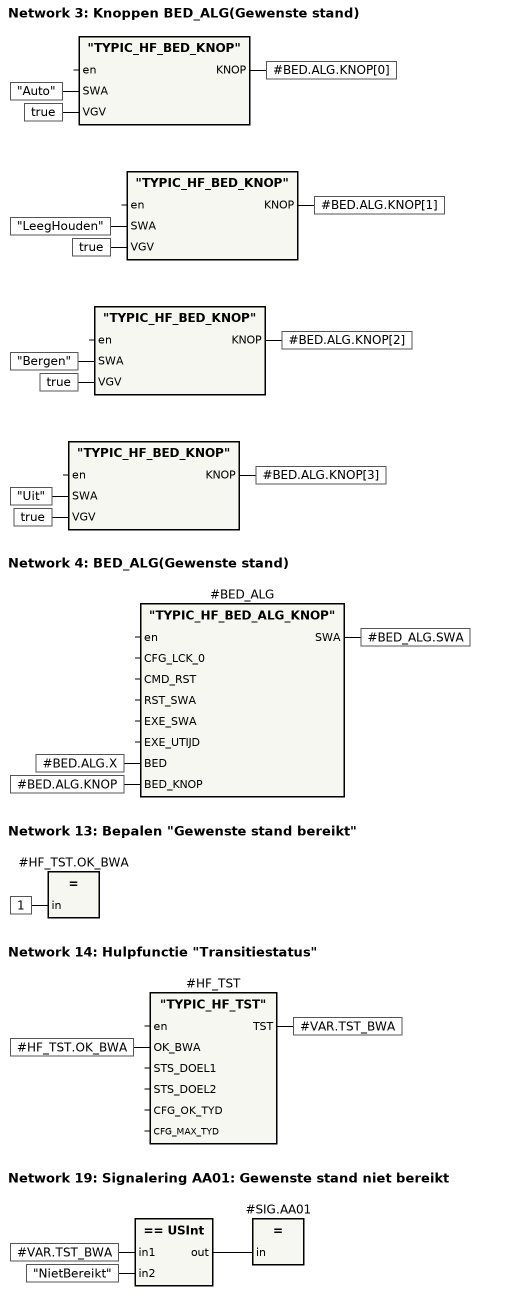
   "TYPIC_HF_BED_KNOP"(SWA := "Auto", VGV := true, KNOP => #BED.ALG.KNOP[0]);
   "TYPIC_HF_BED_KNOP"(SWA := "LeegHouden", VGV := true, KNOP => #BED.ALG.KNOP[1]);
   "TYPIC_HF_BED_KNOP"(SWA := "Bergen", VGV := true, KNOP => #BED.ALG.KNOP[2]);
   "TYPIC_HF_BED_KNOP"(SWA := "Uit", VGV := true, KNOP => #BED.ALG.KNOP[3]);
END_REGION

REGION Network 4: BED_ALG(Gewenste stand)
   // Verwerking BED_ALG
   #BED_ALG(BED := #BED.ALG.X, BED_KNOP := #BED.ALG.KNOP, SWA => #BED_ALG.SWA);   // "TYPIC_HF_BED_ALG_KNOP"
END_REGION

REGION Network 5: +++ Bepalen gewenst regime +++
   // Het gewenst regime (Leeghouden / Bergen / Uit)
END_REGION

REGION Network 6: +++ Bepalen actueel regime en bedieningsmode +++
   // Bepalen bedieningsmode (Automatisch / Manueel / Hand) en
   // 										daarna vastleggen van het actuele regime (Leeghouden /
   // 										Bergen / Uit).
END_REGION

REGION Network 7: +++ Berekeningen +++
   // Verscheidene berekeningen die nodig zijn voor de
   // 										functionele werking of info voor weergave via de centrale en
   // 										lokale bediening, zoals het aantal beschikbare pompen, het
   // 										actueel aantal aangeschakelde pompen en de beschikbare
   // 										pompcapaciteit.
END_REGION

REGION Network 8: +++ Bepalen vloeistofniveau +++
   // Het vloeistofniveau wordt bepaalt door, de status van de
   // 										verschillende vlotters (ontvangen via de niveaumeting) en de
   // 										vlotters droogloopbeveiliging van de pompen, om te zetten
   // 										naar een status.
END_REGION

REGION Network 9: +++ Pompsturing bij regime “Uit” +++
   // Alle pompen behorende tot de schoonvloeistofinstallatie
   // 										worden uitgeschakeld.
END_REGION

REGION Network 10: +++ Pompsturing bij regime “Bergen” +++
   // Pomp(en) aan- of uitschakelen op basis van de peilen LHW
   // 										en HHW van de niveaumeting.
END_REGION

REGION Network 11: +++ Pompsturing bij regime “Leeghouden” +++
   // Pomp(en) aan- of uitschakelen op basis van de peilen SW en
   // 										MSW en LHW van de niveaumeting.
END_REGION

REGION Network 12: +++ Bepalen transitiestatus +++
   // Transitiestatus (bereikt / niet bereikt / in transitie)
   // 										bepalen.
END_REGION

REGION Network 13: Bepalen "Gewenste stand bereikt"
   // Bepalen of de actuele stand in overeenstemming is met de
   // 										gewenste stand
   #HF_TST.OK_BWA := 1;
END_REGION

REGION Network 14: Hulpfunctie "Transitiestatus"
   // De transitiestatus geeft de relatie tussen een gewenste
   // 										stand (van een functionaliteit) en de actuele stand aan.
   #HF_TST(OK_BWA := #HF_TST.OK_BWA, TST => #VAR.TST_BWA);   // "TYPIC_HF_TST"
END_REGION

REGION Network 15: +++ Bepalen beschikbaarheidsstatus +++
   // Beschikbaarheidsstatus (beschikbaar / beperkt beschikbaar
   // 										/ niet beschikbaar) bepalen.
END_REGION

REGION Network 16 (SCL): Beschikbaarheidsstatus bepalen
   IF 
       //voorwaarden "Niet beschikbaar"
       TRUE
   THEN
       //Beschikbaarheidsstatus = Niet Beschikbaar
       #VAR.BSC:= "NietBeschikbaar";
   ELSIF
       //voorwaarden "Beperkt beschikbaar"
       TRUE
   THEN
       //Beschikbaarheidsstatus = Beperkt Beschikbaar
       #VAR.BSC:= "Beperkt";
   ELSE
       //Beschikbaarheidsstatus = Beschikbaar
       #VAR.BSC:= "Beschikbaar";
   END_IF;
END_REGION

REGION Network 17: +++ Signaleringen +++
   // Aanmaken signaleringen.
END_REGION

REGION Network 18 (SCL): Signaleringen voor de onderhoudsoperator
   // Signalering van de storingen ontvangen vanuit de interne
   // 										sturing
   #SIG.A001 := #VAR_IF_SPI.STO.A001;
   #SIG.A002 := #VAR_IF_SPI.STO.A002;
   #SIG.A003 := #VAR_IF_SPI.STO.A003;
   #SIG.A004 := #VAR_IF_SPI.STO.A004;
   #SIG.A005 := #VAR_IF_SPI.STO.A005;
   #SIG.A006 := #VAR_IF_SPI.STO.A006;
   #SIG.A007 := #VAR_IF_SPI.STO.A007;
   #SIG.A008 := #VAR_IF_SPI.STO.A008;
END_REGION

REGION Network 19: Signalering AA01: Gewenste stand niet bereikt
   #SIG.AA01 := #VAR.TST_BWA = "NietBereikt";
END_REGION

REGION Network 20: Signalering AB01 : Niet Beschikbaar
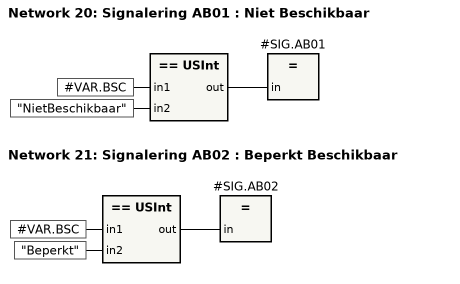
   #SIG.AB01 := #VAR.BSC = "NietBeschikbaar";
END_REGION

REGION Network 21: Signalering AB02 : Beperkt Beschikbaar
   #SIG.AB02 := #VAR.BSC = "Beperkt";
END_REGION

REGION Network 22: +++ Sturingen +++
   // Individuele commandos uitsturen naar iedere pomp om in- en
   // 										uit te schakelen.
END_REGION

REGION Network 23: EINDE
   // Variabelen van intern scada rakvlak naar outputs copieren
END_REGION
END_FUNCTION_BLOCK

FUNCTION_BLOCK "TYPIC_C904_BF_SPI1"   // FB43, FBD
TITLE = TYPIC_C904_BF_SPI1: Schoonvloeistofpompinstallatie
{ S7_Optimized_Access := 'TRUE' }
AUTHOR : OCOTECH
FAMILY : Typical
NAME : C904.801
// Logisch Object Besturing: C904.801
// 
// Het doel van de BF SPI (schoonvloeistofpompinstallatie) is om de algemene sturing te voorzien van de schoonvloeistofpompinstallatie.
// 
// De algemene sturing omvat het weergeven van de algemene toestand en het aano en afschakelen van pompen in functie van het vloeistofpeil en het actieve regime.
// stored: MemoryReserve 10, SetENOAutomatically false
   VAR_INPUT
      CFG_TST_UTYD { ExternalAccessible := 'False'; ExternalVisible := 'False'; ExternalWritable := 'False'} : Time;   // Time-out standverandering pompinstallatie (transitiestatus onbereikt)
      CFG_TST_OK_TYD { ExternalAccessible := 'False'; ExternalVisible := 'False'; ExternalWritable := 'False'} : Time;   // Stabilisatietijd voor de toestand OK (bereikt)
      CFG_NIV_H { ExternalAccessible := 'False'; ExternalVisible := 'False'; ExternalWritable := 'False'} : Real;   // Grenswaarde voor dreigende overloop (minder dan 30m3 bergruimte)
      CFG_NIV_HH { ExternalAccessible := 'False'; ExternalVisible := 'False'; ExternalWritable := 'False'} : Real;   // Grenswaarde voor overloop
      CFG_NIV_ITYD { ExternalAccessible := 'False'; ExternalVisible := 'False'; ExternalWritable := 'False'} : Time;   // Inschakelvertraging storingen grenswaarde
      CFG_NIV_HYS { ExternalAccessible := 'False'; ExternalVisible := 'False'; ExternalWritable := 'False'} : Real;   // Hysteresis storingen grenswaarde
      CFG_DEB_H { ExternalAccessible := 'False'; ExternalVisible := 'False'; ExternalWritable := 'False'} : Real;   // Grenswaarde minimaal debiet bij 1 aangeschakelde pomp
      CFG_DEB_HH { ExternalAccessible := 'False'; ExternalVisible := 'False'; ExternalWritable := 'False'} : Real;   // Grenswaarde minimaal debiet bij meerdere aangeschakelde pompen
      CFG_ITYD_DEB { ExternalAccessible := 'False'; ExternalVisible := 'False'; ExternalWritable := 'False'} : Time;   // Tijdsvertraging voor alarm afvoer verstopt (pomp aangeschakeld en minimaal debiet niet bereikt)
      STU_CMD_AUT { ExternalAccessible := 'False'; ExternalVisible := 'False'; ExternalWritable := 'False'} : USInt;   // Groepscommando: schakel in automatisch
      STU_CMD_WRE { ExternalAccessible := 'False'; ExternalVisible := 'False'; ExternalWritable := 'False'} : USInt;   // Sturing regime
      STU_ALG_LCK_SIG { ExternalAccessible := 'False'; ExternalVisible := 'False'; ExternalWritable := 'False'} : USInt;   // Onderdruk alarmen
   END_VAR
   VAR_OUTPUT
      VAR_PWR { ExternalAccessible := 'False'; ExternalVisible := 'False'; ExternalWritable := 'False'} : Real;   // Som actuele vermogens van alle pompen
      STU_PMP1 { ExternalAccessible := 'False'; ExternalVisible := 'False'; ExternalWritable := 'False'} : USInt;   // Sturing pomp
      STU_PMP2 { ExternalAccessible := 'False'; ExternalVisible := 'False'; ExternalWritable := 'False'} : USInt;   // Sturing pomp
      STU_PMP3 { ExternalAccessible := 'False'; ExternalVisible := 'False'; ExternalWritable := 'False'} : USInt;   // Sturing pomp
      STU_IF_SPI { ExternalAccessible := 'False'; ExternalVisible := 'False'; ExternalWritable := 'False'} : USInt;   // Gewenst regime (naar interne sturing)
   END_VAR
   VAR_IN_OUT
      VAR_IF_SPI : "C904_VAR_IF_SPI_TYPIC";   // Struct met variabelen ontvangen van de interne sturing van de pompinstallatie
      VAR_PMP : Array[*] of "C904_VAR_PMP_TYPIC";   // Array met alle pompen, met alle variabelen van de pomp
      VAR_NIV : "C904_VAR_NIV_TYPIC";   // Struct met alle variabelen ontvangen van de subfunctie niveaumeting
      VAR_DEB : "C904_VAR_DEB_TYPIC";   // Struct met alle variabelen ontvangen van de subfunctie debietmeting
   END_VAR
   VAR
      BED : Struct   // Bedieningen
         ALG : Struct   // Gewenste stand
            X : "UDT_BED_ALG";
            KNOP { S7_SetPoint := 'True'} : Array[0..3] of "UDT_BED_KNOP";
         END_STRUCT;
      END_STRUCT;
      BED_ALG { ExternalWritable := 'False'} : "TYPIC_HF_BED_ALG_KNOP";   // Gewenste stand
      SIG { ExternalWritable := 'False'} : Struct   // Signaleringen
         AA01 : Bool;   // Gewenste stand niet bereikt (transitiestatus = niet bereikt)
         AA02 : Bool;   // Schoonvloeistofpompinstallatie dreigt over te lopen
         AA03 : Bool;   // Overschrijding capaciteit schoonvloeistofpompinstallatie (overloop)
         AA04 : Bool;   // Afvoer verstopt en dreiging overloop van de schoonvloeistofpompinstallatie
         AA05 : Bool;   // Afvoer verstopt
         AB01 : Bool;   // Schoonvloeistofpompinstallatie niet beschikbaar
         AB02 : Bool;   // Schoonvloeistofpompinstallatie beperkt beschikbaar
         A001 : Bool;   // Beveiliging aangesproken
         A002 : Bool;   // Beveiliging No-Break aangesproken
         A003 : Bool;   // Overspanningsbeveiliging aangesproken
         A004 : Bool;   // Schuif ALSB uitgeschakeld
         A005 : Bool;   // Schuif ALSB in test
         A006 : Bool;   // Schuif ALSB uitgereden
         A007 : Bool;   // Nisdeur niet gesloten
         A008 : Bool;   // Storing tracing
      END_STRUCT;
      VAR { ExternalWritable := 'False'} : Struct   // Variabelen
         BSC : USInt;   // Geeft de beschikbaarheid aan van het deelsysteem
         TST_BWA : USInt;   // De status van de transitie van het deelsysteem
         BMO : USInt;   // Bedieningsmode
         WRE_BWA : USInt;   // Actueel regime
         CAPA : USInt;   // Beschikbare pompcapaciteit
         STS_TRA : USInt;   // Status van de tracing
         STS_NIV : USInt;   // Vloeistofniveau bepaald door de stand van de vlotters
         WRE_SWA { ExternalAccessible := 'False'; ExternalVisible := 'False'} : USInt;   // Gewenst regime
         REQ_AAN { ExternalAccessible := 'False'; ExternalVisible := 'False'} : USInt;   // Gewenst aantal aangeschakelde pompen
         CAPA_OK { ExternalAccessible := 'False'; ExternalVisible := 'False'} : USInt;   // Aantal beschikbare pompen
         STS_AAN { ExternalAccessible := 'False'; ExternalVisible := 'False'} : USInt;   // Actueel aantal aangeschakelde pompen
      END_STRUCT;
      HF_TST { ExternalAccessible := 'False'; ExternalVisible := 'False'; ExternalWritable := 'False'} : "TYPIC_HF_TST";   // Hulpfunctie transitiestatus
   END_VAR
   // // BED.ALG.KNOP[0] : Auto
   // // BED.ALG.KNOP[1] : Leeghouden
   // // BED.ALG.KNOP[2] : Bergen
   // // BED.ALG.KNOP[3] : Uit
BEGIN

REGION Network 1: START
END_REGION

REGION Network 2: +++ Bedieningen +++
   // Vrijgave en verwerking van de bedieningen (centrale en lokale bediening). De bedienwaardes worden daarna in de verdere deelfunctionaliteiten gebruikt.
END_REGION

REGION Network 3: Knoppen BED_ALG(Gewenste stand)
   // Waardes en vrijge van de knoppen BED_ALG
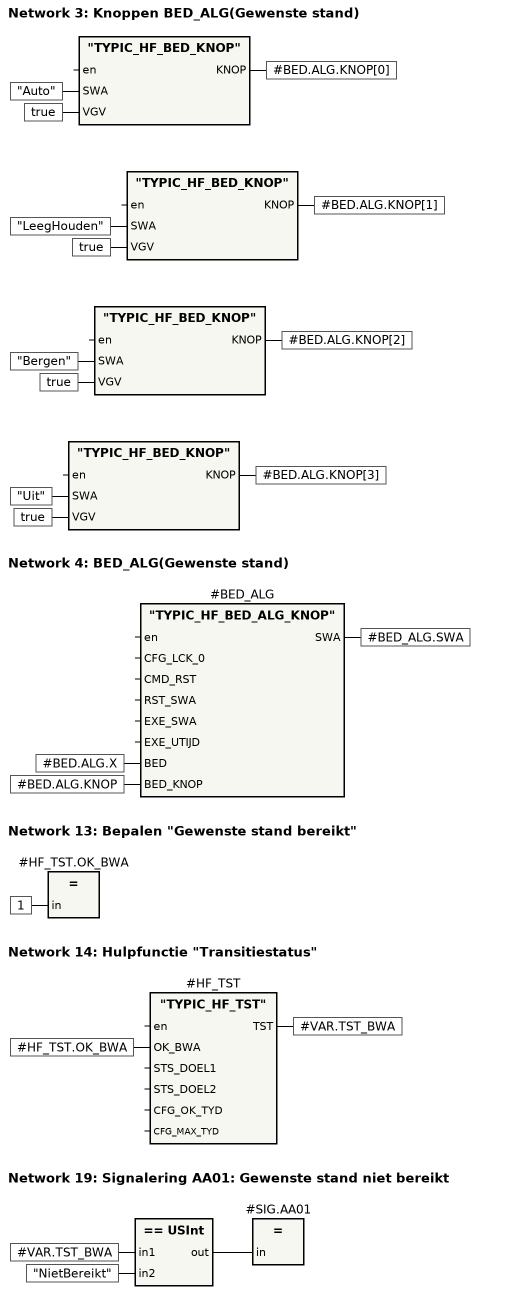
   "TYPIC_HF_BED_KNOP"(SWA := "Auto", VGV := true, KNOP => #BED.ALG.KNOP[0]);
   "TYPIC_HF_BED_KNOP"(SWA := "LeegHouden", VGV := true, KNOP => #BED.ALG.KNOP[1]);
   "TYPIC_HF_BED_KNOP"(SWA := "Bergen", VGV := true, KNOP => #BED.ALG.KNOP[2]);
   "TYPIC_HF_BED_KNOP"(SWA := "Uit", VGV := true, KNOP => #BED.ALG.KNOP[3]);
END_REGION

REGION Network 4: BED_ALG(Gewenste stand)
   // Verwerking BED_ALG
   #BED_ALG(BED := #BED.ALG.X, BED_KNOP := #BED.ALG.KNOP, SWA => #BED_ALG.SWA);   // "TYPIC_HF_BED_ALG_KNOP"
END_REGION

REGION Network 5: +++ Bepalen gewenst regime +++
   // Het gewenst regime (Leeghouden / Bergen / Uit)
END_REGION

REGION Network 6: +++ Bepalen actueel regime en bedieningsmode +++
   // Bepalen bedieningsmode (Automatisch / Manueel / Hand) en daarna vastleggen van het actuele regime (Leeghouden / Bergen / Uit).
END_REGION

REGION Network 7: +++ Berekeningen +++
   // Verscheidene berekeningen die nodig zijn voor de functionele werking of info voor weergave via de centrale en lokale bediening, zoals het aantal beschikbare pompen, het actueel aantal aangeschakelde pompen en de beschikbare pompcapaciteit.
END_REGION

REGION Network 8: +++ Bepalen vloeistofniveau +++
   // Het vloeistofniveau wordt bepaalt door, de status van de verschillende vlotters (ontvangen via de niveaumeting) en de vlotters droogloopbeveiliging van de pompen, om te zetten naar een status.
END_REGION

REGION Network 9: +++ Pompsturing bij regime “Uit” +++
   // Alle pompen behorende tot de schoonvloeistofinstallatie worden uitgeschakeld.
END_REGION

REGION Network 10: +++ Pompsturing bij regime “Bergen” +++
   // Pomp(en) aan- of uitschakelen op basis van de peilen LHW en HHW van de niveaumeting.
END_REGION

REGION Network 11: +++ Pompsturing bij regime “Leeghouden” +++
   // Pomp(en) aan- of uitschakelen op basis van de peilen SW en MSW en LHW van de niveaumeting.
END_REGION

REGION Network 12: +++ Bepalen transitiestatus +++
   // Transitiestatus (bereikt / niet bereikt / in transitie) bepalen.
END_REGION

REGION Network 13: Bepalen "Gewenste stand bereikt"
   // Bepalen of de actuele stand in overeenstemming is met de gewenste stand
   #HF_TST.OK_BWA := 1;
END_REGION

REGION Network 14: Hulpfunctie "Transitiestatus"
   // De transitiestatus geeft de relatie tussen een gewenste stand (van een functionaliteit) en de actuele stand aan.
   #HF_TST(OK_BWA := #HF_TST.OK_BWA, TST => #VAR.TST_BWA);   // "TYPIC_HF_TST"
END_REGION

REGION Network 15: +++ Bepalen beschikbaarheidsstatus +++
   // Beschikbaarheidsstatus (beschikbaar / beperkt beschikbaar / niet beschikbaar) bepalen.
END_REGION

REGION Network 16 (SCL): Beschikbaarheidsstatus bepalen
   IF 
       //voorwaarden "Niet beschikbaar"
       TRUE
   THEN
       //Beschikbaarheidsstatus = Niet Beschikbaar
       #VAR.BSC:= "NietBeschikbaar";
   ELSIF
       //voorwaarden "Beperkt beschikbaar"
       TRUE
   THEN
       //Beschikbaarheidsstatus = Beperkt Beschikbaar
       #VAR.BSC:= "Beperkt";
   ELSE
       //Beschikbaarheidsstatus = Beschikbaar
       #VAR.BSC:= "Beschikbaar";
   END_IF;
END_REGION

REGION Network 17: +++ Signaleringen +++
   // Aanmaken signaleringen.
END_REGION

REGION Network 18 (SCL): Signaleringen voor de onderhoudsoperator
   // Signalering van de storingen ontvangen vanuit de interne sturing
   #SIG.A001 := #VAR_IF_SPI.STO.A001;
   #SIG.A002 := #VAR_IF_SPI.STO.A002;
   #SIG.A003 := #VAR_IF_SPI.STO.A003;
   #SIG.A004 := #VAR_IF_SPI.STO.A004;
   #SIG.A005 := #VAR_IF_SPI.STO.A005;
   #SIG.A006 := #VAR_IF_SPI.STO.A006;
   #SIG.A007 := #VAR_IF_SPI.STO.A007;
   #SIG.A008 := #VAR_IF_SPI.STO.A008;
END_REGION

REGION Network 19: Signalering AA01: Gewenste stand niet bereikt
   #SIG.AA01 := #VAR.TST_BWA = "NietBereikt";
END_REGION

REGION Network 20: Signalering AB01 : Niet Beschikbaar
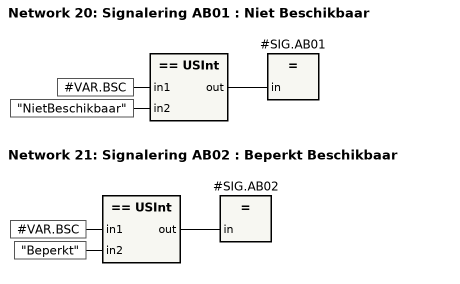
   #SIG.AB01 := #VAR.BSC = "NietBeschikbaar";
END_REGION

REGION Network 21: Signalering AB02 : Beperkt Beschikbaar
   #SIG.AB02 := #VAR.BSC = "Beperkt";
END_REGION

REGION Network 22: +++ Sturingen +++
   // Individuele commandos uitsturen naar iedere pomp om in- en uit te schakelen.
END_REGION

REGION Network 23: EINDE
   // Variabelen van intern scada rakvlak naar outputs copieren
END_REGION
END_FUNCTION_BLOCK

FUNCTION_BLOCK "TYPIC_C904_BF_VPI"   // FB42, FBD
TITLE = TYPIC_C904_BF_VPI: Vuilvloeistofpompinstallatie
{ S7_Optimized_Access := 'TRUE' }
AUTHOR : OCOTECH
FAMILY : Typical
NAME : C904.802
// Logisch Object Besturing: C904.802
// 
// Het doel van de BF VPI (vuilvloeistofpompinstallatie) is om de algemene sturing te voorzien van de vuilvloeistofpompinstallatie.
// 
// De algemene sturing omvat het weergeven van de algemene toestand en het aano en afschakelen van pompen in functie van het vloeistofpeil en het actieve regime.
// stored: MemoryReserve 10, SetENOAutomatically false
   VAR_INPUT
      CFG_TST_UTYD { ExternalAccessible := 'False'; ExternalVisible := 'False'; ExternalWritable := 'False'} : Time;   // Time-out standverandering pompinstallatie (transitiestatus onbereikt)
      CFG_TST_OK_TYD { ExternalAccessible := 'False'; ExternalVisible := 'False'; ExternalWritable := 'False'} : Time;   // Stabilisatietijd voor de toestand OK (bereikt)
      CFG_DEB_H { ExternalAccessible := 'False'; ExternalVisible := 'False'; ExternalWritable := 'False'} : Real;   // Grenswaarde minimaal debiet bij 1 aangeschakelde pomp
      CFG_ITYD_DEB { ExternalAccessible := 'False'; ExternalVisible := 'False'; ExternalWritable := 'False'} : Time;   // Tijdsvertraging voor alarm afvoer verstopt (pomp aangeschakeld en minimaal debiet niet bereikt)
      STU_CMD_AUT { ExternalAccessible := 'False'; ExternalVisible := 'False'; ExternalWritable := 'False'} : USInt;   // Groepscommando: schakel in automatisch
      STU_CMD_WRE { ExternalAccessible := 'False'; ExternalVisible := 'False'; ExternalWritable := 'False'} : USInt;   // Sturing regime
      STU_ALG_LCK_SIG { ExternalAccessible := 'False'; ExternalVisible := 'False'; ExternalWritable := 'False'} : USInt;   // Onderdruk alarmen
   END_VAR
   VAR_OUTPUT
      VAR_PWR { ExternalAccessible := 'False'; ExternalVisible := 'False'; ExternalWritable := 'False'} : Real;   // Som actuele vermogens van alle pompen
      STU_PMP1 { ExternalAccessible := 'False'; ExternalVisible := 'False'; ExternalWritable := 'False'} : USInt;   // Sturing pomp
      STU_PMP2 { ExternalAccessible := 'False'; ExternalVisible := 'False'; ExternalWritable := 'False'} : USInt;   // Sturing pomp
      STU_PMP3 { ExternalAccessible := 'False'; ExternalVisible := 'False'; ExternalWritable := 'False'} : USInt;   // Sturing pomp
      STU_IF_VPI { ExternalAccessible := 'False'; ExternalVisible := 'False'; ExternalWritable := 'False'} : USInt;   // Gewenst regime (naar interne sturing)
   END_VAR
   VAR_IN_OUT
      VAR_IF_VPI : "C904_VAR_IF_VPI_TYPIC";   // Struct met variabelen ontvangen van de interne sturing van de pompinstallatie
      VAR_PMP : Array[*] of "C904_VAR_PMP_TYPIC";   // Array met alle pompen, met alle variabelen van de pomp
      VAR_NIV : "C904_VAR_NIV_TYPIC";   // Struct met alle variabelen ontvangen van de subfunctie niveaumeting
      VAR_DEB : "C904_VAR_DEB_TYPIC";   // Struct met alle variabelen ontvangen van de subfunctie debietmeting
   END_VAR
   VAR
      BED : Struct   // Bedieningen
         ALG : Struct   // Gewenste stand
            X : "UDT_BED_ALG";
            KNOP { S7_SetPoint := 'True'} : Array[0..2] of "UDT_BED_KNOP";
         END_STRUCT;
      END_STRUCT;
      BED_ALG { ExternalWritable := 'False'} : "TYPIC_HF_BED_ALG_KNOP";   // Gewenste stand
      SIG { ExternalWritable := 'False'} : Struct   // Signaleringen
         AA01 : Bool;   // Gewenste stand niet bereikt (transitiestatus = niet bereikt)
         AA02 : Bool;   // Afvoer verstopt
         AB01 : Bool;   // Vuilvloeistofpompinstallatie niet beschikbaar
         AB02 : Bool;   // Vuilvloeistofpompinstallatie beperkt beschikbaar
      END_STRUCT;
      VAR { ExternalWritable := 'False'} : Struct   // Variabelen
         BSC : USInt;   // Geeft de beschikbaarheid aan van het deelsysteem
         TST_BWA : USInt;   // De status van de transitie van het deelsysteem
         BMO : USInt;   // Bedieningsmode
         WRE_BWA : USInt;   // Actueel regime
         CAPA : USInt;   // Beschikbare pompcapaciteit
         STS_NIV : USInt;   // Vloeistofniveau bepaald door de stand van de vlotters
         WRE_SWA { ExternalAccessible := 'False'; ExternalVisible := 'False'} : USInt;   // Gewenst regime
         REQ_AAN { ExternalAccessible := 'False'; ExternalVisible := 'False'} : USInt;   // Gewenst aantal aangeschakelde pompen
         CAPA_OK { ExternalAccessible := 'False'; ExternalVisible := 'False'} : USInt;   // Aantal beschikbare pompen
         STS_AAN { ExternalAccessible := 'False'; ExternalVisible := 'False'} : USInt;   // Actueel aantal aangeschakelde pompen
      END_STRUCT;
      HF_TST { ExternalAccessible := 'False'; ExternalVisible := 'False'; ExternalWritable := 'False'} : "TYPIC_HF_TST";   // Hulpfunctie transitiestatus
   END_VAR
   // // BED.ALG.KNOP[0] : Auto
   // // BED.ALG.KNOP[1] : Lozen
   // // BED.ALG.KNOP[2] : Uit
BEGIN

REGION Network 1: START
END_REGION

REGION Network 2: +++ Bedieningen +++
   // Vrijgave en verwerking van de bedieningen (centrale en lokale bediening). De bedienwaardes worden daarna in de verdere deelfunctionaliteiten gebruikt.
END_REGION

REGION Network 3: Knoppen BED_ALG(Gewenste stand)
   // Waardes en vrijge van de knoppen BED_ALG
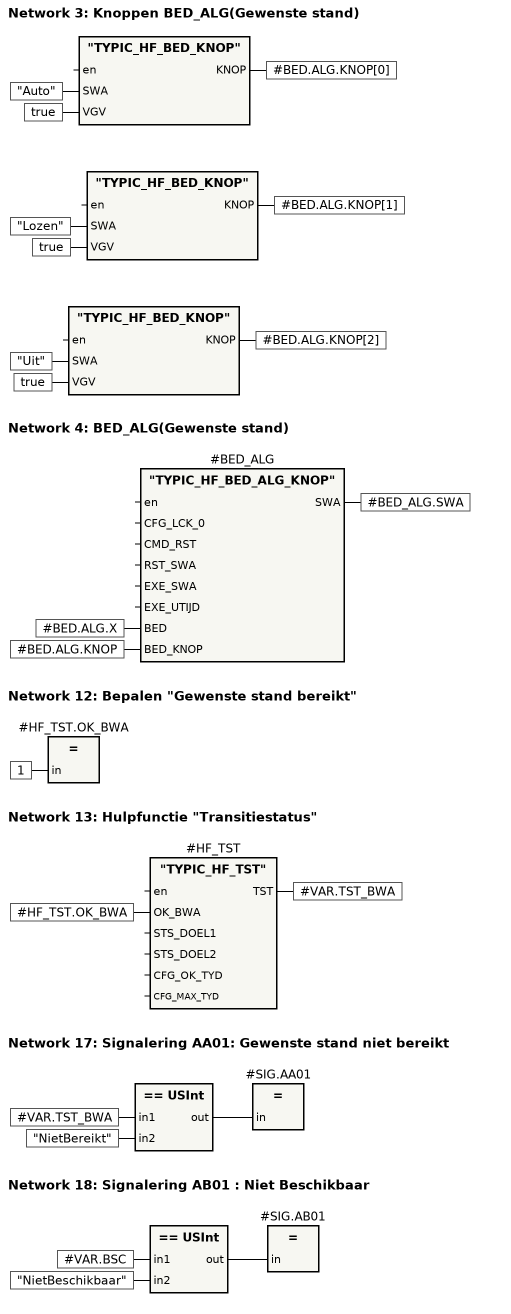
   "TYPIC_HF_BED_KNOP"(SWA := "Auto", VGV := true, KNOP => #BED.ALG.KNOP[0]);
   "TYPIC_HF_BED_KNOP"(SWA := "Lozen", VGV := true, KNOP => #BED.ALG.KNOP[1]);
   "TYPIC_HF_BED_KNOP"(SWA := "Uit", VGV := true, KNOP => #BED.ALG.KNOP[2]);
END_REGION

REGION Network 4: BED_ALG(Gewenste stand)
   // Verwerking BED_ALG
   #BED_ALG(BED := #BED.ALG.X, BED_KNOP := #BED.ALG.KNOP, SWA => #BED_ALG.SWA);   // "TYPIC_HF_BED_ALG_KNOP"
END_REGION

REGION Network 5: +++ Bepalen gewenst regime +++
   // Het gewenst regime (Lozen / Uit)
END_REGION

REGION Network 6: +++ Bepalen actueel regime en bedieningsmode +++
   // Bepalen bedieningsmode (Automatisch / Manueel / Hand) en daarna vastleggen van het actuele regime (Lozen / Uit).
END_REGION

REGION Network 7: +++ Berekeningen +++
   // Verscheidene berekeningen die nodig zijn voor de functionele werking of info voor weergave via de centrale en lokale bediening, zoals het aantal beschikbare pompen, het actueel aantal aangeschakelde pompen en de beschikbare pompcapaciteit.
END_REGION

REGION Network 8: +++ Bepalen vloeistofniveau +++
   // Het vloeistofniveau wordt bepaalt door, de status van de verschillende vlotters (ontvangen via de niveaumeting) en de vlotters droogloopbeveiliging van de pompen, om te zetten naar een status.
END_REGION

REGION Network 9: +++ Pompsturing bij regime “Uit” +++
   // Alle pompen behorende tot de schoonvloeistofinstallatie worden uitgeschakeld.
END_REGION

REGION Network 10: +++ Pompsturing bij regime “Lozen” +++
   // Pomp(en) aan- of uitschakelen op basis van de peilen LW en SW van de niveaumeting.
END_REGION

REGION Network 11: +++ Bepalen transitiestatus +++
   // Transitiestatus (bereikt / niet bereikt / in transitie) bepalen.
END_REGION

REGION Network 12: Bepalen "Gewenste stand bereikt"
   // Bepalen of de actuele stand in overeenstemming is met de gewenste stand
   #HF_TST.OK_BWA := 1;
END_REGION

REGION Network 13: Hulpfunctie "Transitiestatus"
   // De transitiestatus geeft de relatie tussen een gewenste stand (van een functionaliteit) en de actuele stand aan.
   #HF_TST(OK_BWA := #HF_TST.OK_BWA, TST => #VAR.TST_BWA);   // "TYPIC_HF_TST"
END_REGION

REGION Network 14: +++ Bepalen beschikbaarheidsstatus +++
   // Beschikbaarheidsstatus (beschikbaar / beperkt beschikbaar / niet beschikbaar) bepalen.
END_REGION

REGION Network 15 (SCL): Beschikbaarheidsstatus bepalen
   IF 
       //voorwaarden "Niet beschikbaar"
       TRUE
   THEN
       //Beschikbaarheidsstatus = Niet Beschikbaar
       #VAR.BSC:= "NietBeschikbaar";
   ELSIF
       //voorwaarden "Beperkt beschikbaar"
       TRUE
   THEN
       //Beschikbaarheidsstatus = Beperkt Beschikbaar
       #VAR.BSC:= "Beperkt";
   ELSE
       //Beschikbaarheidsstatus = Beschikbaar
       #VAR.BSC:= "Beschikbaar";
   END_IF;
END_REGION

REGION Network 16: +++ Signaleringen +++
   // Aanmaken signaleringen.
END_REGION

REGION Network 17: Signalering AA01: Gewenste stand niet bereikt
   #SIG.AA01 := #VAR.TST_BWA = "NietBereikt";
END_REGION

REGION Network 18: Signalering AB01 : Niet Beschikbaar
   #SIG.AB01 := #VAR.BSC = "NietBeschikbaar";
END_REGION

REGION Network 19: Signalering AB02 : Beperkt Beschikbaar
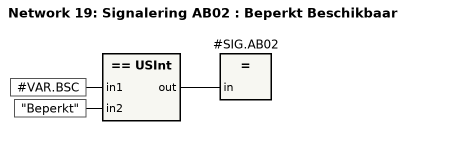
   #SIG.AB02 := #VAR.BSC = "Beperkt";
END_REGION

REGION Network 20: +++ Sturingen +++
   // Individuele commandos uitsturen naar iedere pomp om in- en uit te schakelen.
END_REGION

REGION Network 21: EINDE
   // Variabelen van intern scada rakvlak naar outputs copieren
END_REGION
END_FUNCTION_BLOCK

FUNCTION_BLOCK "TYPIC_C904_IF_SPI"   // FB38, FBD
TITLE = TYPIC_C904_IF_SPI: Schoonvloeistof
{ S7_Optimized_Access := 'TRUE' }
AUTHOR : OCOTECH
FAMILY : Typical
NAME : C904.701
// Logisch Object Besturing: C904.701
// 
// De interne functie schoonvloeistof verzorgt de algemene handbediening via een aanraakscherm.
// stored: MemoryReserve 10, SetENOAutomatically false
   VAR_INPUT
      IN_STS1 { ExternalAccessible := 'False'; ExternalVisible := 'False'; ExternalWritable := 'False'} : Bool;   // Status schuif ALSB in (1 = Ingeschakeld )
      IN_STS2 { ExternalAccessible := 'False'; ExternalVisible := 'False'; ExternalWritable := 'False'} : Bool;   // Status schuif ALSB in test (1 = In Test)
      IN_STS3 { ExternalAccessible := 'False'; ExternalVisible := 'False'; ExternalWritable := 'False'} : Bool;   // Status schuif ALSB uitgereden (1 = Uitgereden)
      IN_NB_AUT { ExternalAccessible := 'False'; ExternalVisible := 'False'; ExternalWritable := 'False'} : Bool;   // Beveiliging No-Break (1 = OK)
      IN_AUT { ExternalAccessible := 'False'; ExternalVisible := 'False'; ExternalWritable := 'False'} : Bool;   // Beveiliging in ALSB-bord (1 = OK)
      IN_KST_TOE { ExternalAccessible := 'False'; ExternalVisible := 'False'; ExternalWritable := 'False'} : Bool;   // Standmelding nisdeur (1 = Toe)
      IN_SPD_OK { ExternalAccessible := 'False'; ExternalVisible := 'False'; ExternalWritable := 'False'} : Bool;   // Status overspanningsbeveiliging (1 = OK)
      IN_TRA_STO { ExternalAccessible := 'False'; ExternalVisible := 'False'; ExternalWritable := 'False'} : Bool;   // Storing tracing (1 = OK / 0 = Storing)
   END_VAR
   VAR_OUTPUT
      VAR_IF_SPI { ExternalAccessible := 'False'; ExternalVisible := 'False'; ExternalWritable := 'False'} : "C904_VAR_IF_SPI_TYPIC";   // Struct met alle variabelen naar bovenliggende functies
   END_VAR
   VAR_IN_OUT
      STU_IF_SPI : USInt;   // Gewenst regime
   END_VAR
   VAR
      BED : Struct   // Bedieningen
         AFSTAND : Bool;   // Bediening om pompinstallatie in afstand te schakelen
         LEEG : Bool;   // Bediening om pompinstallatie in regime Leeghouden te schakelen
         BERG : Bool;   // Bediening om pompinstallatie in regime Bergen te schakelen
         UIT : Bool;   // Bediening om pompinstallatie in regime Uit te schakelen
      END_STRUCT;
      STO { ExternalWritable := 'False'} : Struct   // Storingen
         A001 : Bool;   // Beveiliging aangesproken
         A002 : Bool;   // Beveiliging No-Break aangesproken
         A003 : Bool;   // Overspanningsbeveiliging aangesproken
         A004 : Bool;   // Schuif ALSB uitgeschakeld
         A005 : Bool;   // Schuif ALSB in test
         A006 : Bool;   // Schuif ALSB uitgereden
         A007 : Bool;   // Nisdeur niet gesloten
         A008 : Bool;   // Storing tracing
      END_STRUCT;
      VAR { ExternalWritable := 'False'} : Struct   // Variabelen
         WRE : USInt;   // Actueel actief regime
         BMO_HAND : Bool;   // TRUE = Regime handmatig ingesteld via lokale bediening
      END_STRUCT;
   END_VAR
BEGIN

REGION Network 1: START
END_REGION

REGION Network 2: +++ Bepalen regime en bedieningsmode +++
   // Actueel regime via handbediening instellen en bepalen van de bedieningsmode HAND.
END_REGION

REGION Network 3: +++ Storingen +++
   // Verwerken van de storingsmeldingen (inputs).
END_REGION

REGION Network 4: Storing A001: Beveiliging aangesproken
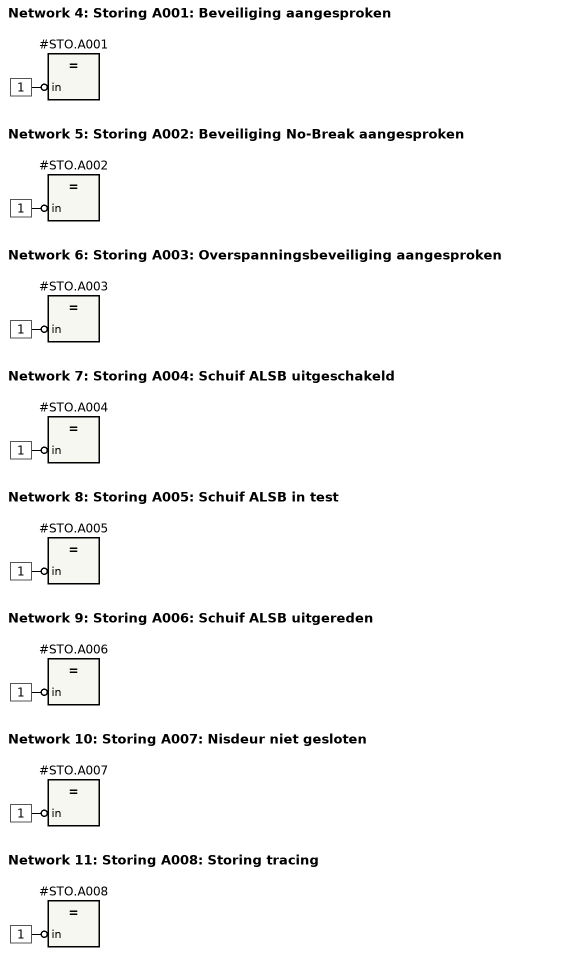
   #STO.A001 := NOT 1;
END_REGION

REGION Network 5: Storing A002: Beveiliging No-Break aangesproken
   #STO.A002 := NOT 1;
END_REGION

REGION Network 6: Storing A003: Overspanningsbeveiliging aangesproken
   #STO.A003 := NOT 1;
END_REGION

REGION Network 7: Storing A004: Schuif ALSB uitgeschakeld
   #STO.A004 := NOT 1;
END_REGION

REGION Network 8: Storing A005: Schuif ALSB in test
   #STO.A005 := NOT 1;
END_REGION

REGION Network 9: Storing A006: Schuif ALSB uitgereden
   #STO.A006 := NOT 1;
END_REGION

REGION Network 10: Storing A007: Nisdeur niet gesloten
   #STO.A007 := NOT 1;
END_REGION

REGION Network 11: Storing A008: Storing tracing
   #STO.A008 := NOT 1;
END_REGION

REGION Network 12 (SCL): EINDE
   // Variabelen van intern scada rakvlak naar outputs copieren
   #VAR_IF_SPI.WRE := #VAR.WRE;
   #VAR_IF_SPI.BMO_HAND := #VAR.BMO_HAND;
   #VAR_IF_SPI.STO := #STO;
END_REGION
END_FUNCTION_BLOCK

FUNCTION_BLOCK "TYPIC_C904_IF_VPI"   // FB37, FBD
TITLE = TYPIC_C904_IF_VPI: Vuilvloeistof
{ S7_Optimized_Access := 'TRUE' }
AUTHOR : OCOTECH
FAMILY : Typical
NAME : C904.702
// Logisch Object Besturing: C904.702
// 
// De interne functie vuilvloeistof verzorgt de algemene handbediening via een aanraakscherm.
// stored: MemoryReserve 10, SetENOAutomatically false
   VAR_OUTPUT
      VAR_IF_VPI { ExternalAccessible := 'False'; ExternalVisible := 'False'; ExternalWritable := 'False'} : "C904_VAR_IF_VPI_TYPIC";   // Struct met alle variabelen naar bovenliggende functies
   END_VAR
   VAR_IN_OUT
      STU_IF_VPI : USInt;   // Gewenst regime
   END_VAR
   VAR
      BED : Struct   // Bedieningen
         AFSTAND : Bool;   // Bediening om pompinstallatie in afstand te schakelen
         LOZ : Bool;   // Bediening om pompinstallatie in regime Lozen te schakelen
         UIT : Bool;   // Bediening om pompinstallatie in regime Uit te schakelen
      END_STRUCT;
      VAR { ExternalWritable := 'False'} : Struct   // Variabelen
         WRE : USInt;   // Actueel actief regime
         BMO_HAND : Bool;   // TRUE = Regime handmatig ingesteld via lokale bediening
      END_STRUCT;
   END_VAR
BEGIN

REGION Network 1: START
END_REGION

REGION Network 2: +++ Bepalen regime en bedieningsmode +++
   // Actueel regime via handbediening instellen en bepalen van de bedieningsmode HAND.
END_REGION

REGION Network 3 (SCL): EINDE
   // Variabelen van intern scada rakvlak naar outputs copieren
   #VAR_IF_VPI.WRE := #VAR.WRE;
   #VAR_IF_VPI.BMO_HAND := #VAR.BMO_HAND;
END_REGION
END_FUNCTION_BLOCK

FUNCTION_BLOCK "TYPIC_C904_SF_PMP"   // FB133, FBD
TITLE = TYPIC_C904_SF_PMP: pomp
{ S7_Optimized_Access := 'TRUE' }
AUTHOR : OCOTECH
FAMILY : Typical
NAME : C904.803
// Logisch Object Besturing: C904.803
// 
// Het doel van deze subfunctie is om de algemene sturing en bediening vanuit 3B te voorzien van een pomp behorende tot de hoofdpompinstallatie.
// stored: MemoryReserve 10, SetENOAutomatically false
   VAR_INPUT
      CFG_PWR { ExternalAccessible := 'False'; ExternalVisible := 'False'; ExternalWritable := 'False'} : Real;   // Nominaal vermogen als pomp aangeschakeld
      STU_CMD_AUT { ExternalAccessible := 'False'; ExternalVisible := 'False'; ExternalWritable := 'False'} : USInt;   // Groepscommando: schakel in automatisch
      STU_ALG_LCK_SIG { ExternalAccessible := 'False'; ExternalVisible := 'False'; ExternalWritable := 'False'} : USInt;   // Onderdruk alarmen
      STU_ENE_VGV_AAN { ExternalAccessible := 'False'; ExternalVisible := 'False'; ExternalWritable := 'False'} : USInt;   // Vrijgeven of verhinderen bijschakelen energieverbruikers (verlichting / ventilatie)
   END_VAR
   VAR_OUTPUT
      VAR_PMP { ExternalAccessible := 'False'; ExternalVisible := 'False'; ExternalWritable := 'False'} : "C904_VAR_PMP_TYPIC";   // Struct met alle variabelen van de pomp
      STU_IF_PMP { ExternalAccessible := 'False'; ExternalVisible := 'False'; ExternalWritable := 'False'} : "C904_STU_IF_PMP_TYPIC";   // Struct met alle sturingen naar de functie (IF) in de interne sturing van de pomp
   END_VAR
   VAR_IN_OUT
      STU_PMP_CMD : USInt;   // Sturing pomp (vanuit de basisfunctie)
      VAR_IF_PMP : "C904_VAR_IF_PMP_TYPIC";   // Struct met alle variabelen van de pomp, ontvangen vanuit de interne sturing
   END_VAR
   VAR
      BED : Struct   // Bedieningen
         ALG : Struct   // Gewenste stand
            X : "UDT_BED_ALG";
            KNOP { S7_SetPoint := 'True'} : Array[0..2] of "UDT_BED_KNOP";
         END_STRUCT;
         BST : Struct   // Bestuurbaarheid
            X : "UDT_BED_ALG";
            KNOP { S7_SetPoint := 'True'} : Array[0..1] of "UDT_BED_KNOP";
         END_STRUCT;
         RES : Struct   // Reset storingen
            X : "UDT_BED_ALG";
            KNOP { S7_SetPoint := 'True'} : Array[0..0] of "UDT_BED_KNOP";
         END_STRUCT;
      END_STRUCT;
      BED_ALG { ExternalWritable := 'False'} : "TYPIC_HF_BED_ALG_KNOP";   // Gewenste stand
      BED_BST { ExternalWritable := 'False'} : "TYPIC_HF_BED_ALG_KNOP";   // Bestuurbaarheid
      BED_RES { ExternalWritable := 'False'} : "TYPIC_HF_BED_ALG_KNOP";   // Reset storingen
      SIG { ExternalWritable := 'False'} : Struct   // Signaleringen
         AA01 : Bool;   // Pomp niet bestuurbaar
         AA02 : Bool;   // Storing algemeen
         A001 : Bool;   // Beveiliging aangesproken
         A002 : Bool;   // Storing van de motorbeveiliging van de pomp
         A003 : Bool;   // Storing motorlade
         A004 : Bool;   // Te hoge temperatuur in de motorwikkelingen
         A005 : Bool;   // Fout stroommeting fase 1
         A006 : Bool;   // Fout stroommeting fase 2
         A007 : Bool;   // Fout stroommeting fase 3
         A008 : Bool;   // Droogloop beveiliging actief: LLW vlotter bovenwater
         A009 : Bool;   // Lekdetectie pomp
         A010 : Bool;   // Motorlade uitgeschakeld
         A011 : Bool;   // Motorlade in test
         A012 : Bool;   // Motorlade uitgereden
         AT01 : Bool;   // Discordantie motor: terugmelding niet ontvangen
         AT02 : Bool;   // Discordantie motor: terugmelding blijft aanwezig
         M001 : Bool;   // Werkschakelaar uitgeschakeld
         M002 : Bool;   // Melding: Pomp heeft te lang niet gedraaid. Periodiek onderhoud nodig
      END_STRUCT;
      VAR { ExternalWritable := 'False'} : Struct   // Variabelen
         TYD_TOT_AAN_UUR : USInt;   // Totaal aantal draaiuren
         ENE_MWA1 : USInt;   // Stroommeting fase 1
         ENE_MWA2 : USInt;   // Stroommeting fase 2
         ENE_MWA3 : USInt;   // Stroommeting fase 3
         RNB : USInt;   // Reden niet bestuurbaar
         AUT : USInt;   // Beveiliging aangesproken
         VGV_SIG_VOP : Bool;   // TRUE = Signaleringen vrijgegeven voor verkeersoperator FALSE = Onderdrukt
         STS : USInt;   // Status van de pomp
         BMO : USInt;   // Bedieningsmode
         BST { ExternalAccessible := 'False'; ExternalVisible := 'False'} : USInt;   // Bestuurbaarheid
         LLW { ExternalAccessible := 'False'; ExternalVisible := 'False'} : USInt;   // Vlotter droogloopbewaking
         PWR { ExternalAccessible := 'False'; ExternalVisible := 'False'} : Real;   // Actueel vermogen van de pomp
         TYD_TOT_AAN { ExternalAccessible := 'False'; ExternalVisible := 'False'} : USInt;   // Totaal aantal draaiuren
         TYD_AAN { ExternalAccessible := 'False'; ExternalVisible := 'False'} : USInt;   // Tijdsduur dat pomp aangeschakeld is
         TYD_UIT { ExternalAccessible := 'False'; ExternalVisible := 'False'} : USInt;   // Tijdsduur dat pomp uitgeschakeld is
      END_STRUCT;
      HF_BST_OBS { ExternalAccessible := 'False'; ExternalVisible := 'False'; ExternalWritable := 'False'} : "TYPIC_HF_BST_OBS";   // Hulp functie besturing
   END_VAR
   // // BED.ALG.KNOP[0] : AUTO
   // // BED.ALG.KNOP[1] : Aan
   // // BED.ALG.KNOP[2] : Uit
   // // BED.BST.KNOP[0] : InDienst
   // // BED.BST.KNOP[1] : UitDienst
   // // BED.RES.KNOP[0] : Reset
BEGIN

REGION Network 1: START
END_REGION

REGION Network 2: +++ Bedieningen +++
   // Vrijgave en verwerking van de bedieningen (centrale en lokale bediening). De bedienwaardes worden daarna in de verdere deelfunctionaliteiten gebruikt.
END_REGION

REGION Network 3: Knoppen BED_ALG(Gewenste stand)
   // Waardes en vrijge van de knoppen BED_ALG
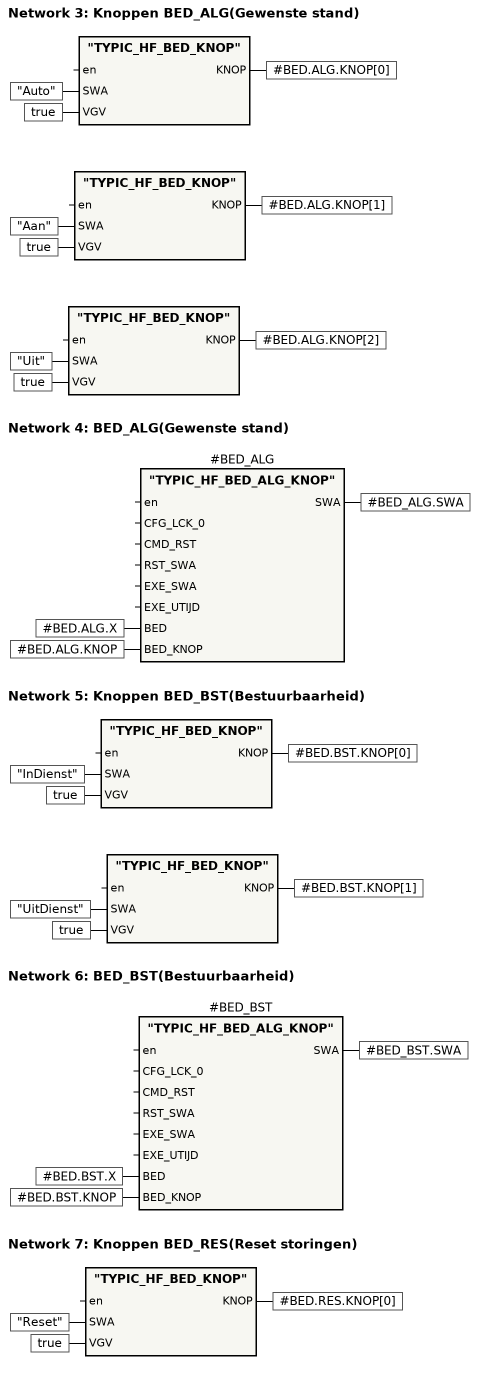
   "TYPIC_HF_BED_KNOP"(SWA := "Auto", VGV := true, KNOP => #BED.ALG.KNOP[0]);
   "TYPIC_HF_BED_KNOP"(SWA := "Aan", VGV := true, KNOP => #BED.ALG.KNOP[1]);
   "TYPIC_HF_BED_KNOP"(SWA := "Uit", VGV := true, KNOP => #BED.ALG.KNOP[2]);
END_REGION

REGION Network 4: BED_ALG(Gewenste stand)
   // Verwerking BED_ALG
   #BED_ALG(BED := #BED.ALG.X, BED_KNOP := #BED.ALG.KNOP, SWA => #BED_ALG.SWA);   // "TYPIC_HF_BED_ALG_KNOP"
END_REGION

REGION Network 5: Knoppen BED_BST(Bestuurbaarheid)
   // Waardes en vrijge van de knoppen BED_BST
   "TYPIC_HF_BED_KNOP"(SWA := "InDienst", VGV := true, KNOP => #BED.BST.KNOP[0]);
   "TYPIC_HF_BED_KNOP"(SWA := "UitDienst", VGV := true, KNOP => #BED.BST.KNOP[1]);
END_REGION

REGION Network 6: BED_BST(Bestuurbaarheid)
   // Verwerking BED_BST
   #BED_BST(BED := #BED.BST.X, BED_KNOP := #BED.BST.KNOP, SWA => #BED_BST.SWA);   // "TYPIC_HF_BED_ALG_KNOP"
END_REGION

REGION Network 7: Knoppen BED_RES(Reset storingen)
   // Waardes en vrijge van de knoppen BED_RES
   "TYPIC_HF_BED_KNOP"(SWA := "Reset", VGV := true, KNOP => #BED.RES.KNOP[0]);
END_REGION

REGION Network 8: BED_RES(Reset storingen)
   // Verwerking BED_RES
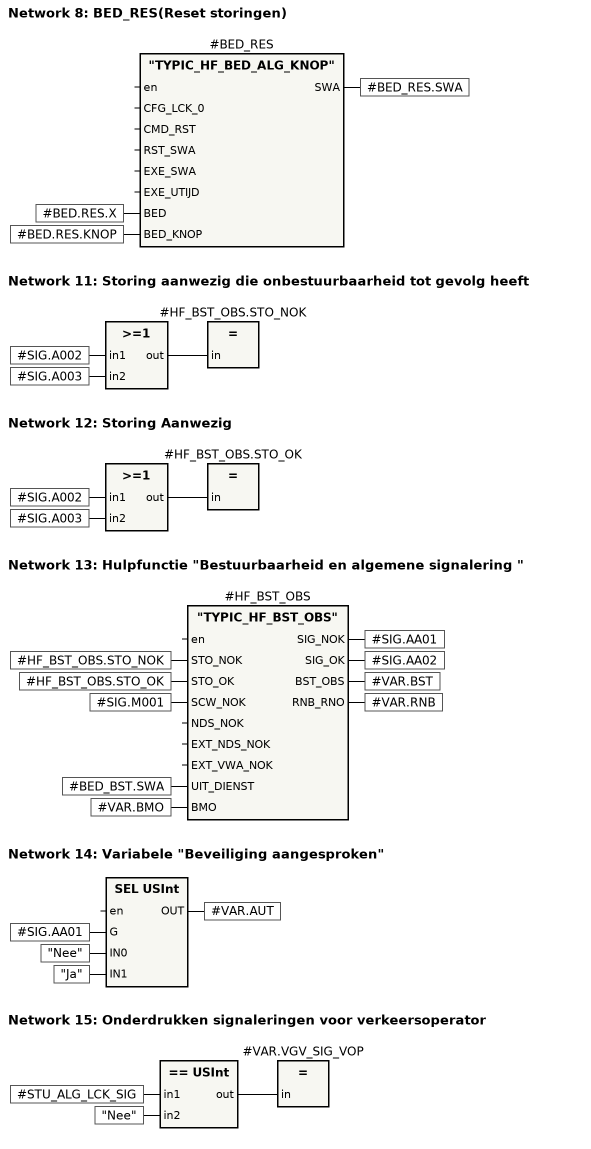
   #BED_RES(BED := #BED.RES.X, BED_KNOP := #BED.RES.KNOP, SWA => #BED_RES.SWA);   // "TYPIC_HF_BED_ALG_KNOP"
END_REGION

REGION Network 9: +++ Bepalen bedieningsmode +++
   // Bedieningsmode (Auto / Manueel / Hand) bepalen.
END_REGION

REGION Network 10: +++ Signaleringen en bestuurbaarheid +++
   // Aanmaken signaleringen, bepalen bestuurbaarheid (bestuurbaar / niet bestuurbaar) en bepalen reden van niet bestuurbaarheid.
END_REGION

REGION Network 11: Storing aanwezig die onbestuurbaarheid tot gevolg heeft
   // OR-verknoping van alle storingen om input STO_BST_NOK van de hulpfunctie "Bestuurbaarheid en algemene signlaring"
   #HF_BST_OBS.STO_NOK := #SIG.A002 OR #SIG.A003;
END_REGION

REGION Network 12: Storing Aanwezig
   // OR-verknoping van alle storingen om input STO_BST_OK van de hulpfunctie "Bestuurbaarheid en algemene signlaring"
   #HF_BST_OBS.STO_OK := #SIG.A002 OR #SIG.A003;
END_REGION

REGION Network 13: Hulpfunctie "Bestuurbaarheid en algemene signalering "
   // Bepalen variabele "bestuurbaarheid" en "reden niet bestuurbaar", Signaleringen "bestuurbaarheid" en "algmene storing".
   #HF_BST_OBS(STO_NOK := #HF_BST_OBS.STO_NOK,   // "TYPIC_HF_BST_OBS"
               STO_OK := #HF_BST_OBS.STO_OK,
               SCW_NOK := #SIG.M001,
               UIT_DIENST := #BED_BST.SWA,
               BMO := #VAR.BMO,
               SIG_NOK => #SIG.AA01,
               SIG_OK => #SIG.AA02,
               BST_OBS => #VAR.BST,
               RNB_RNO => #VAR.RNB);
END_REGION

REGION Network 14: Variabele "Beveiliging aangesproken"
   // De variabele VAR_AUT geef aan of er een beveilliging aangesproken is. Deze variabele laat toe dat de verkeersoperator op SCADA kan zien of er een beveilliging aangesproken is voor deze component.
   #VAR.AUT := SEL(G := #SIG.AA01, IN0 := "Nee", IN1 := "Ja");
END_REGION

REGION Network 15: Onderdrukken signaleringen voor verkeersoperator
   // Via de variabele VGV_SIG_VOP wordt aan IRIS SCADA doorgegeven of signaleringen (bestemd voor de verkeersoperator) van de deze functie zichtbaar (of onderdrukt) moeten zijn.
   #VAR.VGV_SIG_VOP := #STU_ALG_LCK_SIG = "Nee";
END_REGION

REGION Network 16: +++ Bepalen status en actueel vermogen +++
   // Status (Aan / Uit) en actueel verbruikt vermogen bepalen.
END_REGION

REGION Network 17: +++ Draaiuren en fasestromen +++
   // Totaal aantal draaiuren, momentaan aantal draaiuren (actueel aantal uren dat pomp draait / actueel aantal uren dat pomp stilstaat) en fasestromen bepalen.
END_REGION

REGION Network 18: +++ Sturingen +++
   // Commandos naar de interne sturing van de pomp uitsturen.
END_REGION

REGION Network 19 (SCL): EINDE
   // Variabelen van intern scada rakvlak naar outputs copieren
   #VAR_PMP.STS := #VAR.STS;
   #VAR_PMP.BMO := #VAR.BMO;
   #VAR_PMP.BST := #VAR.BST;
   #VAR_PMP.LLW := #VAR.LLW;
   #VAR_PMP.PWR := #VAR.PWR;
   #VAR_PMP.TYD_TOT_AAN := #VAR.TYD_TOT_AAN;
   #VAR_PMP.TYD_AAN := #VAR.TYD_AAN;
   #VAR_PMP.TYD_UIT := #VAR.TYD_UIT;
END_REGION
END_FUNCTION_BLOCK

FUNCTION_BLOCK "TYPIC_C215_IF_PBK"   // FB128, FBD
{ S7_Optimized_Access := 'TRUE' }
AUTHOR : OCOTECH
FAMILY : Typical
NAME : C215.703
// stored: MemoryReserve 10, SetENOAutomatically false
   VAR_INPUT
      EXT_AUT { ExternalAccessible := 'False'; ExternalVisible := 'False'; ExternalWritable := 'False'} : Bool;   // Externe (hoofd) beveiliging (1 = OK)
      EXT_HW { ExternalAccessible := 'False'; ExternalVisible := 'False'; ExternalWritable := 'False'} : Bool;   // Sturings hardware (PLC) bewaking (1 = OK)
      IN_AUT_C215 { ExternalAccessible := 'False'; ExternalVisible := 'False'; ExternalWritable := 'False'} : Bool;   // Serie geschakelde beveiligingen (1 = OK)
      IN_BAT { ExternalAccessible := 'False'; ExternalVisible := 'False'; ExternalWritable := 'False'} : Bool;   // Batterij (1 = OK)
   END_VAR
   VAR_OUTPUT
      VAR_IF_PBK { ExternalAccessible := 'False'; ExternalVisible := 'False'; ExternalWritable := 'False'} : "C215_VAR_IF_PBK_TYPIC";   // Struct met alle variabelen naar bovenliggende functies
   END_VAR
   VAR
      STO { ExternalWritable := 'False'} : Struct   // Storingen
         A001 : Bool;   // Beveiliging aangesproken
         A002 : Bool;   // Storing batterij
      END_STRUCT;
      VAR { ExternalWritable := 'False'} : Struct   // Variabelen
         EXT_AUT { ExternalAccessible := 'False'; ExternalVisible := 'False'} : Bool;   // Externe (hoofd) beveiliging aangesproken
         EXT_HW { ExternalAccessible := 'False'; ExternalVisible := 'False'} : Bool;   // Sturings hardware (PLC) in storing
      END_STRUCT;
   END_VAR
BEGIN
END_FUNCTION_BLOCK

FUNCTION_BLOCK "TYPIC_C215_SF_PBK"   // FB125, FBD
{ S7_Optimized_Access := 'TRUE' }
AUTHOR : OCOTECH
FAMILY : Typical
NAME : C215.804
// stored: MemoryReserve 10, SetENOAutomatically false
   VAR_INPUT
      STU_ALG_LCK_SIG { ExternalAccessible := 'False'; ExternalVisible := 'False'; ExternalWritable := 'False'} : USInt;   // Onderdruk alarmen
   END_VAR
   VAR_IN_OUT
      VAR_IF_PBK : "C215_VAR_IF_PBK_TYPIC";   // Struct met alle variabelen ontvangen van de functie (IF) in de interne sturing van het intern verlicht pictogram kopdeur
   END_VAR
   VAR
      SIG { ExternalWritable := 'False'} : Struct   // Signaleringen
         AA01 : Bool;   // Intern verlicht pictogram kopdeur niet observeerbaar
         AA02 : Bool;   // Algemene storing
         A001 : Bool;   // Beveiliging aangesproken
         A002 : Bool;   // Storing batterij
      END_STRUCT;
      VAR { ExternalWritable := 'False'} : Struct   // Variabelen
         OBS : USInt;   // Observeerbaarheid
         RNO : USInt;   // Reden niet observeerbaar
         AUT : USInt;   // Beveiliging aangesproken
         VGV_SIG_VOP : Bool;   // TRUE = Signaleringen vrijgegeven voor verkeersoperator FALSE = Onderdrukt
      END_STRUCT;
      HF_BST_OBS { ExternalAccessible := 'False'; ExternalVisible := 'False'; ExternalWritable := 'False'} : "TYPIC_HF_BST_OBS";   // Hulp functie besturing
   END_VAR
BEGIN
END_FUNCTION_BLOCK
